BEGIN
	//проверка загруженных данных
	IF #load <> #last THEN
	    #ok := FALSE;
	END_IF;
	
	//первичная загрузка данных
	IF NOT #ok THEN
	    "KP_2_10_DB".KP[0].CMD := "KP_2_10_DB".KP[#load].CMD;
	    "KP_2_10_DB".KP[0].Mode := "KP_2_10_DB".KP[#load].Mode;
	    "KP_2_10_DB".KP[0].Status := "KP_2_10_DB".KP[#load].Status;
	    "KP_2_10_DB".KP[0].FB := "KP_2_10_DB".KP[#load].FB;
	    "KP_2_10_DB".KP[0].Use := "KP_2_10_DB".KP[#load].Use;
	    "KP_2_10_DB".KP[0].Alarm := "KP_2_10_DB".KP[#load].Alarm;
	    "KP_2_10_DB".KP[0].Clock[0].SP := "KP_2_10_DB".KP[#load].Clock[0].SP;
	    "KP_2_10_DB".KP[0].Clock[0].Now := "KP_2_10_DB".KP[#load].Clock[0].Now;
	    "KP_2_10_DB".KP[0].Clock[1].SP := "KP_2_10_DB".KP[#load].Clock[1].SP;
	    "KP_2_10_DB".KP[0].Clock[1].Now := "KP_2_10_DB".KP[#load].Clock[1].Now;
	    "KP_2_10_DB".KP[0].Clock[2].SP := "KP_2_10_DB".KP[#load].Clock[2].SP;
	    "KP_2_10_DB".KP[0].Clock[2].Now := "KP_2_10_DB".KP[#load].Clock[2].Now;
	    "KP_2_10_DB".KP[0].Clock[3].SP := "KP_2_10_DB".KP[#load].Clock[3].SP;
	    "KP_2_10_DB".KP[0].Clock[3].Now := "KP_2_10_DB".KP[#load].Clock[3].Now;
	    "KP_2_10_DB".KP[0].Clock[4].SP := "KP_2_10_DB".KP[#load].Clock[4].SP;
	    "KP_2_10_DB".KP[0].Clock[4].Now := "KP_2_10_DB".KP[#load].Clock[4].Now;
	    "KP_2_10_DB".KP[0].CodeID := "KP_2_10_DB".KP[#load].CodeID;
	    "KP_2_10_DB".KP[0].Position := "KP_2_10_DB".KP[#load].Position;
	    "KP_2_10_DB".KP[0].Speed := "KP_2_10_DB".KP[#load].Speed;
	    "KP_2_10_DB".KP[0].Name := "KP_2_10_DB".KP[#load].Name;
	    #ok := true;
	    #last := #load;
	END_IF;
	
	//управление с панели
	IF #ok THEN
	    "KP_2_10_DB".KP[#load].CMD.Hand := "KP_2_10_DB".KP[0].CMD.Hand;
	    "KP_2_10_DB".KP[#load].CMD.Force := "KP_2_10_DB".KP[0].CMD.Force;
	    "KP_2_10_DB".KP[#load].CMD.Start_M := "KP_2_10_DB".KP[0].CMD.Start_M;
	    "KP_2_10_DB".KP[#load].CMD.Reset := "KP_2_10_DB".KP[0].CMD.Reset;
	    "KP_2_10_DB".KP[#load].Use := "KP_2_10_DB".KP[0].Use;
	    "KP_2_10_DB".KP[#load].Clock[0].SP := "KP_2_10_DB".KP[0].Clock[0].SP;
	    "KP_2_10_DB".KP[#load].Clock[1].SP := "KP_2_10_DB".KP[0].Clock[1].SP;
	    "KP_2_10_DB".KP[#load].Clock[2].SP := "KP_2_10_DB".KP[0].Clock[2].SP;
	    "KP_2_10_DB".KP[#load].Clock[3].SP := "KP_2_10_DB".KP[0].Clock[3].SP;
	    "KP_2_10_DB".KP[#load].Clock[4].SP := "KP_2_10_DB".KP[0].Clock[4].SP;
	    "KP_2_10_DB".KP[#load].CodeID := "KP_2_10_DB".KP[0].CodeID;
	    "KP_2_10_DB".KP[#load].Speed := "KP_2_10_DB".KP[0].Speed;
	    "KP_2_10_DB".KP[0].CMD.Local := "KP_2_10_DB".KP[#load].CMD.Local;
	    "KP_2_10_DB".KP[0].CMD.Lock := "KP_2_10_DB".KP[#load].CMD.Lock;
	    "KP_2_10_DB".KP[0].Mode := "KP_2_10_DB".KP[#load].Mode;
	    "KP_2_10_DB".KP[0].Status := "KP_2_10_DB".KP[#load].Status;
	    "KP_2_10_DB".KP[0].FB := "KP_2_10_DB".KP[#load].FB;
	    "KP_2_10_DB".KP[0].Alarm := "KP_2_10_DB".KP[#load].Alarm;
	    "KP_2_10_DB".KP[0].Clock[0].Now := "KP_2_10_DB".KP[#load].Clock[0].Now;
	    "KP_2_10_DB".KP[0].Clock[1].Now := "KP_2_10_DB".KP[#load].Clock[1].Now;
	    "KP_2_10_DB".KP[0].Clock[2].Now := "KP_2_10_DB".KP[#load].Clock[2].Now;
	    "KP_2_10_DB".KP[0].Clock[3].Now := "KP_2_10_DB".KP[#load].Clock[3].Now;
	    "KP_2_10_DB".KP[0].Clock[4].Now := "KP_2_10_DB".KP[#load].Clock[4].Now;
	    "KP_2_10_DB".KP[0].Position := "KP_2_10_DB".KP[#load].Position;
	    IF "KP_2_10_DB".KP[0].CMD.Reset THEN
	        "KP_2_10_DB".KP[0].CMD.Reset := FALSE;
	    END_IF;
	END_IF;
	
	    
END_FUNCTION

FUNCTION_BLOCK "KP_1"
{ S7_Optimized_Access := 'FALSE' }
VERSION : 0.1
   VAR 
      limit { S7_SetPoint := 'True'} : Int := 2;   // число задвижек в камере
      load : Int;   // отображаемые на экране настройки
      load_last : Int;
      KP : Array[0..10] of "DRV_AUMA";
      load_ok { S7_SetPoint := 'True'} : Bool;
   END_VAR

   VAR_TEMP 
      ID : Int;
      cnt : Int;
   END_VAR


BEGIN
	
	"Load_KP_1"(last := #load_last,
	              load := #load,
	              ok := #load_ok);
	  IF "KP_Reset" THEN
	      #load := 10;
	  END_IF;
	
	FOR #cnt := 1 TO #limit BY 1 DO
	    #ID := #KP[#cnt].CodeID;
	    #KP[#cnt].CMD.Local := NOT "AUMA_KP_1_DB".AUMA[#ID].Message.Sel_Dist;
	    #KP[#cnt].Alarm.Link := NOT "AUMA_KP_1_DB".AUMA[#ID].Link;
	    #KP[#cnt].Use.Enable := "AUMA_KP_1_DB".AUMA[#ID].Use;
	    #KP[#cnt].Name := "AUMA_KP_1_DB".AUMA[#ID].Name;
	    #KP[#cnt].Position := INT_TO_REAL("AUMA_KP_1_DB".AUMA[#ID].Position) / 10.0;
	    #KP[#cnt].FB.QF := "AUMA_KP_1_DB".AUMA[#ID].Message.NotReady;
	    #KP[#cnt].FB.KM_Open := "AUMA_KP_1_DB".AUMA[#ID].Message.Opening;
	    #KP[#cnt].FB.KM_Close := "AUMA_KP_1_DB".AUMA[#ID].Message.Closing;
	    #KP[#cnt].FB.Open := "AUMA_KP_1_DB".AUMA[#ID].Message.Open;
	    #KP[#cnt].FB.Close := "AUMA_KP_1_DB".AUMA[#ID].Message.Close;
	    #KP[#cnt]();
	    "AUMA_KP_1_DB".AUMA[#ID].Speed := #KP[#cnt].Speed;
	    "AUMA_KP_1_DB".AUMA[#ID].CMD.Open := #KP[#cnt].CMD_Open;
	    "AUMA_KP_1_DB".AUMA[#ID].CMD.Close := #KP[#cnt].CMD_Close;
	    IF "AUMA_KP_1_DB".AUMA[#ID].CMD.Open <> "AUMA_KP_1_DB".AUMA[#ID].CMD_last.Open THEN
	        "AUMA_KP_1_DB".AUMA[#ID].CMD_last.Open := "AUMA_KP_1_DB".AUMA[#ID].CMD.Open;
	        "AUMA_KP_1_DB".AUMA[#ID].Update := true;
	    END_IF;
	    IF "AUMA_KP_1_DB".AUMA[#ID].CMD.Close <> "AUMA_KP_1_DB".AUMA[#ID].CMD_last.Close THEN
	        "AUMA_KP_1_DB".AUMA[#ID].CMD_last.Close := "AUMA_KP_1_DB".AUMA[#ID].CMD.Close;
	        "AUMA_KP_1_DB".AUMA[#ID].Update := true;
	    END_IF;
	END_FOR;
END_FUNCTION_BLOCK

FUNCTION "Load_KP_1" : Void
{ S7_Optimized_Access := 'TRUE' }
VERSION : 0.1
   VAR_IN_OUT 
      ok : Bool;
      load : Int;
      last : Int;
   END_VAR


BEGIN
	//проверка загруженных данных
	IF #load <> #last THEN
	    #ok := FALSE;
	END_IF;
	
	//первичная загрузка данных
	IF NOT #ok THEN
	    "KP_1_DB".KP[0].CMD := "KP_1_DB".KP[#load].CMD;
	    "KP_1_DB".KP[0].Mode := "KP_1_DB".KP[#load].Mode;
	    "KP_1_DB".KP[0].Status := "KP_1_DB".KP[#load].Status;
	    "KP_1_DB".KP[0].FB := "KP_1_DB".KP[#load].FB;
	    "KP_1_DB".KP[0].Use := "KP_1_DB".KP[#load].Use;
	    "KP_1_DB".KP[0].Alarm := "KP_1_DB".KP[#load].Alarm;
	    "KP_1_DB".KP[0].Clock[0].SP := "KP_1_DB".KP[#load].Clock[0].SP;
	    "KP_1_DB".KP[0].Clock[0].Now := "KP_1_DB".KP[#load].Clock[0].Now;
	    "KP_1_DB".KP[0].Clock[1].SP := "KP_1_DB".KP[#load].Clock[1].SP;
	    "KP_1_DB".KP[0].Clock[1].Now := "KP_1_DB".KP[#load].Clock[1].Now;
	    "KP_1_DB".KP[0].Clock[2].SP := "KP_1_DB".KP[#load].Clock[2].SP;
	    "KP_1_DB".KP[0].Clock[2].Now := "KP_1_DB".KP[#load].Clock[2].Now;
	    "KP_1_DB".KP[0].Clock[3].SP := "KP_1_DB".KP[#load].Clock[3].SP;
	    "KP_1_DB".KP[0].Clock[3].Now := "KP_1_DB".KP[#load].Clock[3].Now;
	    "KP_1_DB".KP[0].Clock[4].SP := "KP_1_DB".KP[#load].Clock[4].SP;
	    "KP_1_DB".KP[0].Clock[4].Now := "KP_1_DB".KP[#load].Clock[4].Now;
	    "KP_1_DB".KP[0].CodeID := "KP_1_DB".KP[#load].CodeID;
	    "KP_1_DB".KP[0].Position := "KP_1_DB".KP[#load].Position;
	    "KP_1_DB".KP[0].Speed := "KP_1_DB".KP[#load].Speed;
	    "KP_1_DB".KP[0].Name := "KP_1_DB".KP[#load].Name;
	    #ok := true;
	    #last := #load;
	END_IF;
	
	//управление с панели
	IF #ok THEN
	    "KP_1_DB".KP[#load].CMD.Hand := "KP_1_DB".KP[0].CMD.Hand;
	    "KP_1_DB".KP[#load].CMD.Force := "KP_1_DB".KP[0].CMD.Force;
	    "KP_1_DB".KP[#load].CMD.Start_M := "KP_1_DB".KP[0].CMD.Start_M;
	    "KP_1_DB".KP[#load].CMD.Reset := "KP_1_DB".KP[0].CMD.Reset;
	    "KP_1_DB".KP[#load].Use := "KP_1_DB".KP[0].Use;
	    "KP_1_DB".KP[#load].Clock[0].SP := "KP_1_DB".KP[0].Clock[0].SP;
	    "KP_1_DB".KP[#load].Clock[1].SP := "KP_1_DB".KP[0].Clock[1].SP;
	    "KP_1_DB".KP[#load].Clock[2].SP := "KP_1_DB".KP[0].Clock[2].SP;
	    "KP_1_DB".KP[#load].Clock[3].SP := "KP_1_DB".KP[0].Clock[3].SP;
	    "KP_1_DB".KP[#load].Clock[4].SP := "KP_1_DB".KP[0].Clock[4].SP;
	    "KP_1_DB".KP[#load].CodeID := "KP_1_DB".KP[0].CodeID;
	    "KP_1_DB".KP[#load].Speed := "KP_1_DB".KP[0].Speed;
	    "KP_1_DB".KP[0].CMD.Local := "KP_1_DB".KP[#load].CMD.Local;
	    "KP_1_DB".KP[0].CMD.Lock := "KP_1_DB".KP[#load].CMD.Lock;
	    "KP_1_DB".KP[0].Mode := "KP_1_DB".KP[#load].Mode;
	    "KP_1_DB".KP[0].Status := "KP_1_DB".KP[#load].Status;
	    "KP_1_DB".KP[0].FB := "KP_1_DB".KP[#load].FB;
	    "KP_1_DB".KP[0].Alarm := "KP_1_DB".KP[#load].Alarm;
	    "KP_1_DB".KP[0].Clock[0].Now := "KP_1_DB".KP[#load].Clock[0].Now;
	    "KP_1_DB".KP[0].Clock[1].Now := "KP_1_DB".KP[#load].Clock[1].Now;
	    "KP_1_DB".KP[0].Clock[2].Now := "KP_1_DB".KP[#load].Clock[2].Now;
	    "KP_1_DB".KP[0].Clock[3].Now := "KP_1_DB".KP[#load].Clock[3].Now;
	    "KP_1_DB".KP[0].Clock[4].Now := "KP_1_DB".KP[#load].Clock[4].Now;
	    "KP_1_DB".KP[0].Position := "KP_1_DB".KP[#load].Position;
	    IF "KP_1_DB".KP[0].CMD.Reset THEN
	        "KP_1_DB".KP[0].CMD.Reset := FALSE;
	    END_IF;
	END_IF;
	
	    
END_FUNCTION

FUNCTION_BLOCK "KP_2"
{ S7_Optimized_Access := 'FALSE' }
VERSION : 0.1
   VAR 
      limit { S7_SetPoint := 'True'} : Int := 2;   // число задвижек в камере
      load : Int;   // отображаемые на экране настройки
      load_last : Int;
      KP : Array[0..10] of "DRV_AUMA";
      load_ok { S7_SetPoint := 'True'} : Bool;
   END_VAR

   VAR_TEMP 
      ID : Int;
      cnt : Int;
   END_VAR


BEGIN
	
	"Load_KP_2"(last := #load_last,
	              load := #load,
	              ok := #load_ok);
	  IF "KP_Reset" THEN
	      #load := 10;
	  END_IF;
	
	FOR #cnt := 1 TO #limit BY 1 DO
	    #ID := #KP[#cnt].CodeID;
	    #KP[#cnt].CMD.Local := NOT "AUMA_KP_2_DB".AUMA[#ID].Message.Sel_Dist;
	    #KP[#cnt].Alarm.Link := NOT "AUMA_KP_2_DB".AUMA[#ID].Link;
	    #KP[#cnt].Use.Enable := "AUMA_KP_2_DB".AUMA[#ID].Use;
	    #KP[#cnt].Name := "AUMA_KP_2_DB".AUMA[#ID].Name;
	    #KP[#cnt].Position := INT_TO_REAL("AUMA_KP_2_DB".AUMA[#ID].Position) / 10.0;
	    #KP[#cnt].FB.QF := "AUMA_KP_2_DB".AUMA[#ID].Message.NotReady;
	    #KP[#cnt].FB.KM_Open := "AUMA_KP_2_DB".AUMA[#ID].Message.Opening;
	    #KP[#cnt].FB.KM_Close := "AUMA_KP_2_DB".AUMA[#ID].Message.Closing;
	    #KP[#cnt].FB.Open := "AUMA_KP_2_DB".AUMA[#ID].Message.Open;
	    #KP[#cnt].FB.Close := "AUMA_KP_2_DB".AUMA[#ID].Message.Close;
	    #KP[#cnt]();
	    "AUMA_KP_2_DB".AUMA[#ID].Speed := #KP[#cnt].Speed;
	    "AUMA_KP_2_DB".AUMA[#ID].CMD.Open := #KP[#cnt].CMD_Open;
	    "AUMA_KP_2_DB".AUMA[#ID].CMD.Close := #KP[#cnt].CMD_Close;
	    IF "AUMA_KP_2_DB".AUMA[#ID].CMD.Open <> "AUMA_KP_2_DB".AUMA[#ID].CMD_last.Open THEN
	        "AUMA_KP_2_DB".AUMA[#ID].CMD_last.Open := "AUMA_KP_2_DB".AUMA[#ID].CMD.Open;
	        "AUMA_KP_2_DB".AUMA[#ID].Update := true;
	    END_IF;
	    IF "AUMA_KP_2_DB".AUMA[#ID].CMD.Close <> "AUMA_KP_2_DB".AUMA[#ID].CMD_last.Close THEN
	        "AUMA_KP_2_DB".AUMA[#ID].CMD_last.Close := "AUMA_KP_2_DB".AUMA[#ID].CMD.Close;
	        "AUMA_KP_2_DB".AUMA[#ID].Update := true;
	    END_IF;
	END_FOR;
END_FUNCTION_BLOCK

FUNCTION "Load_KP_2" : Void
{ S7_Optimized_Access := 'TRUE' }
VERSION : 0.1
   VAR_IN_OUT 
      ok : Bool;
      load : Int;
      last : Int;
   END_VAR


BEGIN
	//проверка загруженных данных
	IF #load <> #last THEN
	    #ok := FALSE;
	END_IF;
	
	//первичная загрузка данных
	IF NOT #ok THEN
	    "KP_2_DB".KP[0].CMD := "KP_2_DB".KP[#load].CMD;
	    "KP_2_DB".KP[0].Mode := "KP_2_DB".KP[#load].Mode;
	    "KP_2_DB".KP[0].Status := "KP_2_DB".KP[#load].Status;
	    "KP_2_DB".KP[0].FB := "KP_2_DB".KP[#load].FB;
	    "KP_2_DB".KP[0].Use := "KP_2_DB".KP[#load].Use;
	    "KP_2_DB".KP[0].Alarm := "KP_2_DB".KP[#load].Alarm;
	    "KP_2_DB".KP[0].Clock[0].SP := "KP_2_DB".KP[#load].Clock[0].SP;
	    "KP_2_DB".KP[0].Clock[0].Now := "KP_2_DB".KP[#load].Clock[0].Now;
	    "KP_2_DB".KP[0].Clock[1].SP := "KP_2_DB".KP[#load].Clock[1].SP;
	    "KP_2_DB".KP[0].Clock[1].Now := "KP_2_DB".KP[#load].Clock[1].Now;
	    "KP_2_DB".KP[0].Clock[2].SP := "KP_2_DB".KP[#load].Clock[2].SP;
	    "KP_2_DB".KP[0].Clock[2].Now := "KP_2_DB".KP[#load].Clock[2].Now;
	    "KP_2_DB".KP[0].Clock[3].SP := "KP_2_DB".KP[#load].Clock[3].SP;
	    "KP_2_DB".KP[0].Clock[3].Now := "KP_2_DB".KP[#load].Clock[3].Now;
	    "KP_2_DB".KP[0].Clock[4].SP := "KP_2_DB".KP[#load].Clock[4].SP;
	    "KP_2_DB".KP[0].Clock[4].Now := "KP_2_DB".KP[#load].Clock[4].Now;
	    "KP_2_DB".KP[0].CodeID := "KP_2_DB".KP[#load].CodeID;
	    "KP_2_DB".KP[0].Position := "KP_2_DB".KP[#load].Position;
	    "KP_2_DB".KP[0].Speed := "KP_2_DB".KP[#load].Speed;
	    "KP_2_DB".KP[0].Name := "KP_2_DB".KP[#load].Name;
	    #ok := true;
	    #last := #load;
	END_IF;
	
	//управление с панели
	IF #ok THEN
	    "KP_2_DB".KP[#load].CMD.Hand := "KP_2_DB".KP[0].CMD.Hand;
	    "KP_2_DB".KP[#load].CMD.Force := "KP_2_DB".KP[0].CMD.Force;
	    "KP_2_DB".KP[#load].CMD.Start_M := "KP_2_DB".KP[0].CMD.Start_M;
	    "KP_2_DB".KP[#load].CMD.Reset := "KP_2_DB".KP[0].CMD.Reset;
	    "KP_2_DB".KP[#load].Use := "KP_2_DB".KP[0].Use;
	    "KP_2_DB".KP[#load].Clock[0].SP := "KP_2_DB".KP[0].Clock[0].SP;
	    "KP_2_DB".KP[#load].Clock[1].SP := "KP_2_DB".KP[0].Clock[1].SP;
	    "KP_2_DB".KP[#load].Clock[2].SP := "KP_2_DB".KP[0].Clock[2].SP;
	    "KP_2_DB".KP[#load].Clock[3].SP := "KP_2_DB".KP[0].Clock[3].SP;
	    "KP_2_DB".KP[#load].Clock[4].SP := "KP_2_DB".KP[0].Clock[4].SP;
	    "KP_2_DB".KP[#load].CodeID := "KP_2_DB".KP[0].CodeID;
	    "KP_2_DB".KP[#load].Speed := "KP_2_DB".KP[0].Speed;
	    "KP_2_DB".KP[0].CMD.Local := "KP_2_DB".KP[#load].CMD.Local;
	    "KP_2_DB".KP[0].CMD.Lock := "KP_2_DB".KP[#load].CMD.Lock;
	    "KP_2_DB".KP[0].Mode := "KP_2_DB".KP[#load].Mode;
	    "KP_2_DB".KP[0].Status := "KP_2_DB".KP[#load].Status;
	    "KP_2_DB".KP[0].FB := "KP_2_DB".KP[#load].FB;
	    "KP_2_DB".KP[0].Alarm := "KP_2_DB".KP[#load].Alarm;
	    "KP_2_DB".KP[0].Clock[0].Now := "KP_2_DB".KP[#load].Clock[0].Now;
	    "KP_2_DB".KP[0].Clock[1].Now := "KP_2_DB".KP[#load].Clock[1].Now;
	    "KP_2_DB".KP[0].Clock[2].Now := "KP_2_DB".KP[#load].Clock[2].Now;
	    "KP_2_DB".KP[0].Clock[3].Now := "KP_2_DB".KP[#load].Clock[3].Now;
	    "KP_2_DB".KP[0].Clock[4].Now := "KP_2_DB".KP[#load].Clock[4].Now;
	    "KP_2_DB".KP[0].Position := "KP_2_DB".KP[#load].Position;
	    IF "KP_2_DB".KP[0].CMD.Reset THEN
	        "KP_2_DB".KP[0].CMD.Reset := FALSE;
	    END_IF;
	END_IF;
	
	    
END_FUNCTION

FUNCTION_BLOCK "KP_3"
{ S7_Optimized_Access := 'FALSE' }
VERSION : 0.1
   VAR 
      limit { S7_SetPoint := 'True'} : Int := 2;   // число задвижек в камере
      load : Int;   // отображаемые на экране настройки
      load_last : Int;
      KP : Array[0..10] of "DRV_AUMA";
      load_ok { S7_SetPoint := 'True'} : Bool;
   END_VAR

   VAR_TEMP 
      ID : Int;
      cnt : Int;
   END_VAR


BEGIN
	
	"Load_KP_3"(last := #load_last,
	              load := #load,
	              ok := #load_ok);
	  IF "KP_Reset" THEN
	      #load := 10;
	  END_IF;
	
	FOR #cnt := 1 TO #limit BY 1 DO
	    #ID := #KP[#cnt].CodeID;
	    #KP[#cnt].CMD.Local := NOT "AUMA_KP_3_DB".AUMA[#ID].Message.Sel_Dist;
	    #KP[#cnt].Alarm.Link := NOT "AUMA_KP_3_DB".AUMA[#ID].Link;
	    #KP[#cnt].Use.Enable := "AUMA_KP_3_DB".AUMA[#ID].Use;
	    #KP[#cnt].Name := "AUMA_KP_3_DB".AUMA[#ID].Name;
	    #KP[#cnt].Position := INT_TO_REAL("AUMA_KP_3_DB".AUMA[#ID].Position) / 10.0;
	    #KP[#cnt].FB.QF := "AUMA_KP_3_DB".AUMA[#ID].Message.NotReady;
	    #KP[#cnt].FB.KM_Open := "AUMA_KP_3_DB".AUMA[#ID].Message.Opening;
	    #KP[#cnt].FB.KM_Close := "AUMA_KP_3_DB".AUMA[#ID].Message.Closing;
	    #KP[#cnt].FB.Open := "AUMA_KP_3_DB".AUMA[#ID].Message.Open;
	    #KP[#cnt].FB.Close := "AUMA_KP_3_DB".AUMA[#ID].Message.Close;
	    #KP[#cnt]();
	    "AUMA_KP_3_DB".AUMA[#ID].Speed := #KP[#cnt].Speed;
	    "AUMA_KP_3_DB".AUMA[#ID].CMD.Open := #KP[#cnt].CMD_Open;
	    "AUMA_KP_3_DB".AUMA[#ID].CMD.Close := #KP[#cnt].CMD_Close;
	    IF "AUMA_KP_3_DB".AUMA[#ID].CMD.Open <> "AUMA_KP_3_DB".AUMA[#ID].CMD_last.Open THEN
	        "AUMA_KP_3_DB".AUMA[#ID].CMD_last.Open := "AUMA_KP_3_DB".AUMA[#ID].CMD.Open;
	        "AUMA_KP_3_DB".AUMA[#ID].Update := true;
	    END_IF;
	    IF "AUMA_KP_3_DB".AUMA[#ID].CMD.Close <> "AUMA_KP_3_DB".AUMA[#ID].CMD_last.Close THEN
	        "AUMA_KP_3_DB".AUMA[#ID].CMD_last.Close := "AUMA_KP_3_DB".AUMA[#ID].CMD.Close;
	        "AUMA_KP_3_DB".AUMA[#ID].Update := true;
	    END_IF;
	END_FOR;
END_FUNCTION_BLOCK

FUNCTION "Load_KP_3" : Void
{ S7_Optimized_Access := 'TRUE' }
VERSION : 0.1
   VAR_IN_OUT 
      ok : Bool;
      load : Int;
      last : Int;
   END_VAR


BEGIN
	//проверка загруженных данных
	IF #load <> #last THEN
	    #ok := FALSE;
	END_IF;
	
	//первичная загрузка данных
	IF NOT #ok THEN
	    "KP_3_DB".KP[0].CMD := "KP_3_DB".KP[#load].CMD;
	    "KP_3_DB".KP[0].Mode := "KP_3_DB".KP[#load].Mode;
	    "KP_3_DB".KP[0].Status := "KP_3_DB".KP[#load].Status;
	    "KP_3_DB".KP[0].FB := "KP_3_DB".KP[#load].FB;
	    "KP_3_DB".KP[0].Use := "KP_3_DB".KP[#load].Use;
	    "KP_3_DB".KP[0].Alarm := "KP_3_DB".KP[#load].Alarm;
	    "KP_3_DB".KP[0].Clock[0].SP := "KP_3_DB".KP[#load].Clock[0].SP;
	    "KP_3_DB".KP[0].Clock[0].Now := "KP_3_DB".KP[#load].Clock[0].Now;
	    "KP_3_DB".KP[0].Clock[1].SP := "KP_3_DB".KP[#load].Clock[1].SP;
	    "KP_3_DB".KP[0].Clock[1].Now := "KP_3_DB".KP[#load].Clock[1].Now;
	    "KP_3_DB".KP[0].Clock[2].SP := "KP_3_DB".KP[#load].Clock[2].SP;
	    "KP_3_DB".KP[0].Clock[2].Now := "KP_3_DB".KP[#load].Clock[2].Now;
	    "KP_3_DB".KP[0].Clock[3].SP := "KP_3_DB".KP[#load].Clock[3].SP;
	    "KP_3_DB".KP[0].Clock[3].Now := "KP_3_DB".KP[#load].Clock[3].Now;
	    "KP_3_DB".KP[0].Clock[4].SP := "KP_3_DB".KP[#load].Clock[4].SP;
	    "KP_3_DB".KP[0].Clock[4].Now := "KP_3_DB".KP[#load].Clock[4].Now;
	    "KP_3_DB".KP[0].CodeID := "KP_3_DB".KP[#load].CodeID;
	    "KP_3_DB".KP[0].Position := "KP_3_DB".KP[#load].Position;
	    "KP_3_DB".KP[0].Speed := "KP_3_DB".KP[#load].Speed;
	    "KP_3_DB".KP[0].Name := "KP_3_DB".KP[#load].Name;
	    #ok := true;
	    #last := #load;
	END_IF;
	
	//управление с панели
	IF #ok THEN
	    "KP_3_DB".KP[#load].CMD.Hand := "KP_3_DB".KP[0].CMD.Hand;
	    "KP_3_DB".KP[#load].CMD.Force := "KP_3_DB".KP[0].CMD.Force;
	    "KP_3_DB".KP[#load].CMD.Start_M := "KP_3_DB".KP[0].CMD.Start_M;
	    "KP_3_DB".KP[#load].CMD.Reset := "KP_3_DB".KP[0].CMD.Reset;
	    "KP_3_DB".KP[#load].Use := "KP_3_DB".KP[0].Use;
	    "KP_3_DB".KP[#load].Clock[0].SP := "KP_3_DB".KP[0].Clock[0].SP;
	    "KP_3_DB".KP[#load].Clock[1].SP := "KP_3_DB".KP[0].Clock[1].SP;
	    "KP_3_DB".KP[#load].Clock[2].SP := "KP_3_DB".KP[0].Clock[2].SP;
	    "KP_3_DB".KP[#load].Clock[3].SP := "KP_3_DB".KP[0].Clock[3].SP;
	    "KP_3_DB".KP[#load].Clock[4].SP := "KP_3_DB".KP[0].Clock[4].SP;
	    "KP_3_DB".KP[#load].CodeID := "KP_3_DB".KP[0].CodeID;
	    "KP_3_DB".KP[#load].Speed := "KP_3_DB".KP[0].Speed;
	    "KP_3_DB".KP[0].CMD.Local := "KP_3_DB".KP[#load].CMD.Local;
	    "KP_3_DB".KP[0].CMD.Lock := "KP_3_DB".KP[#load].CMD.Lock;
	    "KP_3_DB".KP[0].Mode := "KP_3_DB".KP[#load].Mode;
	    "KP_3_DB".KP[0].Status := "KP_3_DB".KP[#load].Status;
	    "KP_3_DB".KP[0].FB := "KP_3_DB".KP[#load].FB;
	    "KP_3_DB".KP[0].Alarm := "KP_3_DB".KP[#load].Alarm;
	    "KP_3_DB".KP[0].Clock[0].Now := "KP_3_DB".KP[#load].Clock[0].Now;
	    "KP_3_DB".KP[0].Clock[1].Now := "KP_3_DB".KP[#load].Clock[1].Now;
	    "KP_3_DB".KP[0].Clock[2].Now := "KP_3_DB".KP[#load].Clock[2].Now;
	    "KP_3_DB".KP[0].Clock[3].Now := "KP_3_DB".KP[#load].Clock[3].Now;
	    "KP_3_DB".KP[0].Clock[4].Now := "KP_3_DB".KP[#load].Clock[4].Now;
	    "KP_3_DB".KP[0].Position := "KP_3_DB".KP[#load].Position;
	    IF "KP_3_DB".KP[0].CMD.Reset THEN
	        "KP_3_DB".KP[0].CMD.Reset := FALSE;
	    END_IF;
	END_IF;
	
	    
END_FUNCTION

FUNCTION_BLOCK "KP_4"
{ S7_Optimized_Access := 'FALSE' }
VERSION : 0.1
   VAR 
      limit { S7_SetPoint := 'True'} : Int := 2;   // число задвижек в камере
      load : Int;   // отображаемые на экране настройки
      load_last : Int;
      KP : Array[0..10] of "DRV_AUMA";
      load_ok { S7_SetPoint := 'True'} : Bool;
   END_VAR

   VAR_TEMP 
      ID : Int;
      cnt : Int;
   END_VAR


BEGIN
	
	"Load_KP_4"(last := #load_last,
	              load := #load,
	              ok := #load_ok);
	  IF "KP_Reset" THEN
	      #load := 10;
	  END_IF;
	
	FOR #cnt := 1 TO #limit BY 1 DO
	    #ID := #KP[#cnt].CodeID;
	    #KP[#cnt].CMD.Local := NOT "AUMA_KP_4_DB".AUMA[#ID].Message.Sel_Dist;
	    #KP[#cnt].Alarm.Link := NOT "AUMA_KP_4_DB".AUMA[#ID].Link;
	    #KP[#cnt].Use.Enable := "AUMA_KP_4_DB".AUMA[#ID].Use;
	    #KP[#cnt].Name := "AUMA_KP_4_DB".AUMA[#ID].Name;
	    #KP[#cnt].Position := INT_TO_REAL("AUMA_KP_4_DB".AUMA[#ID].Position) / 10.0;
	    #KP[#cnt].FB.QF := "AUMA_KP_4_DB".AUMA[#ID].Message.NotReady;
	    #KP[#cnt].FB.KM_Open := "AUMA_KP_4_DB".AUMA[#ID].Message.Opening;
	    #KP[#cnt].FB.KM_Close := "AUMA_KP_4_DB".AUMA[#ID].Message.Closing;
	    #KP[#cnt].FB.Open := "AUMA_KP_4_DB".AUMA[#ID].Message.Open;
	    #KP[#cnt].FB.Close := "AUMA_KP_4_DB".AUMA[#ID].Message.Close;
	    #KP[#cnt]();
	    "AUMA_KP_4_DB".AUMA[#ID].Speed := #KP[#cnt].Speed;
	    "AUMA_KP_4_DB".AUMA[#ID].CMD.Open := #KP[#cnt].CMD_Open;
	    "AUMA_KP_4_DB".AUMA[#ID].CMD.Close := #KP[#cnt].CMD_Close;
	    IF "AUMA_KP_4_DB".AUMA[#ID].CMD.Open <> "AUMA_KP_4_DB".AUMA[#ID].CMD_last.Open THEN
	        "AUMA_KP_4_DB".AUMA[#ID].CMD_last.Open := "AUMA_KP_4_DB".AUMA[#ID].CMD.Open;
	        "AUMA_KP_4_DB".AUMA[#ID].Update := true;
	    END_IF;
	    IF "AUMA_KP_4_DB".AUMA[#ID].CMD.Close <> "AUMA_KP_4_DB".AUMA[#ID].CMD_last.Close THEN
	        "AUMA_KP_4_DB".AUMA[#ID].CMD_last.Close := "AUMA_KP_4_DB".AUMA[#ID].CMD.Close;
	        "AUMA_KP_4_DB".AUMA[#ID].Update := true;
	    END_IF;
	END_FOR;
END_FUNCTION_BLOCK

FUNCTION "Load_KP_4" : Void
{ S7_Optimized_Access := 'TRUE' }
VERSION : 0.1
   VAR_IN_OUT 
      ok : Bool;
      load : Int;
      last : Int;
   END_VAR


BEGIN
	//проверка загруженных данных
	IF #load <> #last THEN
	    #ok := FALSE;
	END_IF;
	
	//первичная загрузка данных
	IF NOT #ok THEN
	    "KP_4_DB".KP[0].CMD := "KP_4_DB".KP[#load].CMD;
	    "KP_4_DB".KP[0].Mode := "KP_4_DB".KP[#load].Mode;
	    "KP_4_DB".KP[0].Status := "KP_4_DB".KP[#load].Status;
	    "KP_4_DB".KP[0].FB := "KP_4_DB".KP[#load].FB;
	    "KP_4_DB".KP[0].Use := "KP_4_DB".KP[#load].Use;
	    "KP_4_DB".KP[0].Alarm := "KP_4_DB".KP[#load].Alarm;
	    "KP_4_DB".KP[0].Clock[0].SP := "KP_4_DB".KP[#load].Clock[0].SP;
	    "KP_4_DB".KP[0].Clock[0].Now := "KP_4_DB".KP[#load].Clock[0].Now;
	    "KP_4_DB".KP[0].Clock[1].SP := "KP_4_DB".KP[#load].Clock[1].SP;
	    "KP_4_DB".KP[0].Clock[1].Now := "KP_4_DB".KP[#load].Clock[1].Now;
	    "KP_4_DB".KP[0].Clock[2].SP := "KP_4_DB".KP[#load].Clock[2].SP;
	    "KP_4_DB".KP[0].Clock[2].Now := "KP_4_DB".KP[#load].Clock[2].Now;
	    "KP_4_DB".KP[0].Clock[3].SP := "KP_4_DB".KP[#load].Clock[3].SP;
	    "KP_4_DB".KP[0].Clock[3].Now := "KP_4_DB".KP[#load].Clock[3].Now;
	    "KP_4_DB".KP[0].Clock[4].SP := "KP_4_DB".KP[#load].Clock[4].SP;
	    "KP_4_DB".KP[0].Clock[4].Now := "KP_4_DB".KP[#load].Clock[4].Now;
	    "KP_4_DB".KP[0].CodeID := "KP_4_DB".KP[#load].CodeID;
	    "KP_4_DB".KP[0].Position := "KP_4_DB".KP[#load].Position;
	    "KP_4_DB".KP[0].Speed := "KP_4_DB".KP[#load].Speed;
	    "KP_4_DB".KP[0].Name := "KP_4_DB".KP[#load].Name;
	    #ok := true;
	    #last := #load;
	END_IF;
	
	//управление с панели
	IF #ok THEN
	    "KP_4_DB".KP[#load].CMD.Hand := "KP_4_DB".KP[0].CMD.Hand;
	    "KP_4_DB".KP[#load].CMD.Force := "KP_4_DB".KP[0].CMD.Force;
	    "KP_4_DB".KP[#load].CMD.Start_M := "KP_4_DB".KP[0].CMD.Start_M;
	    "KP_4_DB".KP[#load].CMD.Reset := "KP_4_DB".KP[0].CMD.Reset;
	    "KP_4_DB".KP[#load].Use := "KP_4_DB".KP[0].Use;
	    "KP_4_DB".KP[#load].Clock[0].SP := "KP_4_DB".KP[0].Clock[0].SP;
	    "KP_4_DB".KP[#load].Clock[1].SP := "KP_4_DB".KP[0].Clock[1].SP;
	    "KP_4_DB".KP[#load].Clock[2].SP := "KP_4_DB".KP[0].Clock[2].SP;
	    "KP_4_DB".KP[#load].Clock[3].SP := "KP_4_DB".KP[0].Clock[3].SP;
	    "KP_4_DB".KP[#load].Clock[4].SP := "KP_4_DB".KP[0].Clock[4].SP;
	    "KP_4_DB".KP[#load].CodeID := "KP_4_DB".KP[0].CodeID;
	    "KP_4_DB".KP[#load].Speed := "KP_4_DB".KP[0].Speed;
	    "KP_4_DB".KP[0].CMD.Local := "KP_4_DB".KP[#load].CMD.Local;
	    "KP_4_DB".KP[0].CMD.Lock := "KP_4_DB".KP[#load].CMD.Lock;
	    "KP_4_DB".KP[0].Mode := "KP_4_DB".KP[#load].Mode;
	    "KP_4_DB".KP[0].Status := "KP_4_DB".KP[#load].Status;
	    "KP_4_DB".KP[0].FB := "KP_4_DB".KP[#load].FB;
	    "KP_4_DB".KP[0].Alarm := "KP_4_DB".KP[#load].Alarm;
	    "KP_4_DB".KP[0].Clock[0].Now := "KP_4_DB".KP[#load].Clock[0].Now;
	    "KP_4_DB".KP[0].Clock[1].Now := "KP_4_DB".KP[#load].Clock[1].Now;
	    "KP_4_DB".KP[0].Clock[2].Now := "KP_4_DB".KP[#load].Clock[2].Now;
	    "KP_4_DB".KP[0].Clock[3].Now := "KP_4_DB".KP[#load].Clock[3].Now;
	    "KP_4_DB".KP[0].Clock[4].Now := "KP_4_DB".KP[#load].Clock[4].Now;
	    "KP_4_DB".KP[0].Position := "KP_4_DB".KP[#load].Position;
	    IF "KP_4_DB".KP[0].CMD.Reset THEN
	        "KP_4_DB".KP[0].CMD.Reset := FALSE;
	    END_IF;
	END_IF;
	
	    
END_FUNCTION

FUNCTION_BLOCK "KP_5"
{ S7_Optimized_Access := 'FALSE' }
VERSION : 0.1
   VAR 
      limit { S7_SetPoint := 'True'} : Int := 2;   // число задвижек в камере
      load : Int;   // отображаемые на экране настройки
      load_last : Int;
      KP : Array[0..10] of "DRV_AUMA";
      load_ok { S7_SetPoint := 'True'} : Bool;
   END_VAR

   VAR_TEMP 
      ID : Int;
      cnt : Int;
   END_VAR


BEGIN
	
	"Load_KP_5"(last := #load_last,
	              load := #load,
	              ok := #load_ok);
	  IF "KP_Reset" THEN
	      #load := 10;
	  END_IF;
	
	FOR #cnt := 1 TO #limit BY 1 DO
	    #ID := #KP[#cnt].CodeID;
	    #KP[#cnt].CMD.Local := NOT "AUMA_KP_5_DB".AUMA[#ID].Message.Sel_Dist;
	    #KP[#cnt].Alarm.Link := NOT "AUMA_KP_5_DB".AUMA[#ID].Link;
	    #KP[#cnt].Use.Enable := "AUMA_KP_5_DB".AUMA[#ID].Use;
	    #KP[#cnt].Name := "AUMA_KP_5_DB".AUMA[#ID].Name;
	    #KP[#cnt].Position := INT_TO_REAL("AUMA_KP_5_DB".AUMA[#ID].Position) / 10.0;
	    #KP[#cnt].FB.QF := "AUMA_KP_5_DB".AUMA[#ID].Message.NotReady;
	    #KP[#cnt].FB.KM_Open := "AUMA_KP_5_DB".AUMA[#ID].Message.Opening;
	    #KP[#cnt].FB.KM_Close := "AUMA_KP_5_DB".AUMA[#ID].Message.Closing;
	    #KP[#cnt].FB.Open := "AUMA_KP_5_DB".AUMA[#ID].Message.Open;
	    #KP[#cnt].FB.Close := "AUMA_KP_5_DB".AUMA[#ID].Message.Close;
	    #KP[#cnt]();
	    "AUMA_KP_5_DB".AUMA[#ID].Speed := #KP[#cnt].Speed;
	    "AUMA_KP_5_DB".AUMA[#ID].CMD.Open := #KP[#cnt].CMD_Open;
	    "AUMA_KP_5_DB".AUMA[#ID].CMD.Close := #KP[#cnt].CMD_Close;
	    IF "AUMA_KP_5_DB".AUMA[#ID].CMD.Open <> "AUMA_KP_5_DB".AUMA[#ID].CMD_last.Open THEN
	        "AUMA_KP_5_DB".AUMA[#ID].CMD_last.Open := "AUMA_KP_5_DB".AUMA[#ID].CMD.Open;
	        "AUMA_KP_5_DB".AUMA[#ID].Update := true;
	    END_IF;
	    IF "AUMA_KP_5_DB".AUMA[#ID].CMD.Close <> "AUMA_KP_5_DB".AUMA[#ID].CMD_last.Close THEN
	        "AUMA_KP_5_DB".AUMA[#ID].CMD_last.Close := "AUMA_KP_5_DB".AUMA[#ID].CMD.Close;
	        "AUMA_KP_5_DB".AUMA[#ID].Update := true;
	    END_IF;
	END_FOR;
END_FUNCTION_BLOCK

FUNCTION "Load_KP_5" : Void
{ S7_Optimized_Access := 'TRUE' }
VERSION : 0.1
   VAR_IN_OUT 
      ok : Bool;
      load : Int;
      last : Int;
   END_VAR


BEGIN
	//проверка загруженных данных
	IF #load <> #last THEN
	    #ok := FALSE;
	END_IF;
	
	//первичная загрузка данных
	IF NOT #ok THEN
	    "KP_5_DB".KP[0].CMD := "KP_5_DB".KP[#load].CMD;
	    "KP_5_DB".KP[0].Mode := "KP_5_DB".KP[#load].Mode;
	    "KP_5_DB".KP[0].Status := "KP_5_DB".KP[#load].Status;
	    "KP_5_DB".KP[0].FB := "KP_5_DB".KP[#load].FB;
	    "KP_5_DB".KP[0].Use := "KP_5_DB".KP[#load].Use;
	    "KP_5_DB".KP[0].Alarm := "KP_5_DB".KP[#load].Alarm;
	    "KP_5_DB".KP[0].Clock[0].SP := "KP_5_DB".KP[#load].Clock[0].SP;
	    "KP_5_DB".KP[0].Clock[0].Now := "KP_5_DB".KP[#load].Clock[0].Now;
	    "KP_5_DB".KP[0].Clock[1].SP := "KP_5_DB".KP[#load].Clock[1].SP;
	    "KP_5_DB".KP[0].Clock[1].Now := "KP_5_DB".KP[#load].Clock[1].Now;
	    "KP_5_DB".KP[0].Clock[2].SP := "KP_5_DB".KP[#load].Clock[2].SP;
	    "KP_5_DB".KP[0].Clock[2].Now := "KP_5_DB".KP[#load].Clock[2].Now;
	    "KP_5_DB".KP[0].Clock[3].SP := "KP_5_DB".KP[#load].Clock[3].SP;
	    "KP_5_DB".KP[0].Clock[3].Now := "KP_5_DB".KP[#load].Clock[3].Now;
	    "KP_5_DB".KP[0].Clock[4].SP := "KP_5_DB".KP[#load].Clock[4].SP;
	    "KP_5_DB".KP[0].Clock[4].Now := "KP_5_DB".KP[#load].Clock[4].Now;
	    "KP_5_DB".KP[0].CodeID := "KP_5_DB".KP[#load].CodeID;
	    "KP_5_DB".KP[0].Position := "KP_5_DB".KP[#load].Position;
	    "KP_5_DB".KP[0].Speed := "KP_5_DB".KP[#load].Speed;
	    "KP_5_DB".KP[0].Name := "KP_5_DB".KP[#load].Name;
	    #ok := true;
	    #last := #load;
	END_IF;
	
	//управление с панели
	IF #ok THEN
	    "KP_5_DB".KP[#load].CMD.Hand := "KP_5_DB".KP[0].CMD.Hand;
	    "KP_5_DB".KP[#load].CMD.Force := "KP_5_DB".KP[0].CMD.Force;
	    "KP_5_DB".KP[#load].CMD.Start_M := "KP_5_DB".KP[0].CMD.Start_M;
	    "KP_5_DB".KP[#load].CMD.Reset := "KP_5_DB".KP[0].CMD.Reset;
	    "KP_5_DB".KP[#load].Use := "KP_5_DB".KP[0].Use;
	    "KP_5_DB".KP[#load].Clock[0].SP := "KP_5_DB".KP[0].Clock[0].SP;
	    "KP_5_DB".KP[#load].Clock[1].SP := "KP_5_DB".KP[0].Clock[1].SP;
	    "KP_5_DB".KP[#load].Clock[2].SP := "KP_5_DB".KP[0].Clock[2].SP;
	    "KP_5_DB".KP[#load].Clock[3].SP := "KP_5_DB".KP[0].Clock[3].SP;
	    "KP_5_DB".KP[#load].Clock[4].SP := "KP_5_DB".KP[0].Clock[4].SP;
	    "KP_5_DB".KP[#load].CodeID := "KP_5_DB".KP[0].CodeID;
	    "KP_5_DB".KP[#load].Speed := "KP_5_DB".KP[0].Speed;
	    "KP_5_DB".KP[0].CMD.Local := "KP_5_DB".KP[#load].CMD.Local;
	    "KP_5_DB".KP[0].CMD.Lock := "KP_5_DB".KP[#load].CMD.Lock;
	    "KP_5_DB".KP[0].Mode := "KP_5_DB".KP[#load].Mode;
	    "KP_5_DB".KP[0].Status := "KP_5_DB".KP[#load].Status;
	    "KP_5_DB".KP[0].FB := "KP_5_DB".KP[#load].FB;
	    "KP_5_DB".KP[0].Alarm := "KP_5_DB".KP[#load].Alarm;
	    "KP_5_DB".KP[0].Clock[0].Now := "KP_5_DB".KP[#load].Clock[0].Now;
	    "KP_5_DB".KP[0].Clock[1].Now := "KP_5_DB".KP[#load].Clock[1].Now;
	    "KP_5_DB".KP[0].Clock[2].Now := "KP_5_DB".KP[#load].Clock[2].Now;
	    "KP_5_DB".KP[0].Clock[3].Now := "KP_5_DB".KP[#load].Clock[3].Now;
	    "KP_5_DB".KP[0].Clock[4].Now := "KP_5_DB".KP[#load].Clock[4].Now;
	    "KP_5_DB".KP[0].Position := "KP_5_DB".KP[#load].Position;
	    IF "KP_5_DB".KP[0].CMD.Reset THEN
	        "KP_5_DB".KP[0].CMD.Reset := FALSE;
	    END_IF;
	END_IF;
	
	    
END_FUNCTION

FUNCTION_BLOCK "PIDx"   // FB260, LAD
{ S7_Optimized_Access := 'TRUE' }
VERSION : 0.1
// stored: AutoNumber false, IsIECCheckEnabled false, IsRetainMemResEnabled false, MemoryReserve 100, SetENOAutomatically false, UDAEnableTagReadback false
   VAR DB_SPECIFIC
      Time_DTL { S7_SetPoint := 'True'} : DTL;
   END_VAR
BEGIN

REGION Network 2: Метка времени
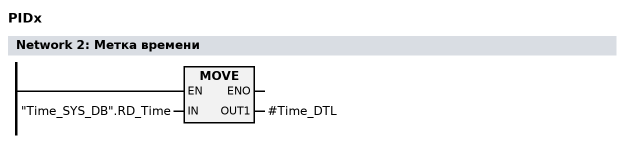
   RUNG wire#powerrail
      Move(in := "Time_SYS_DB".RD_Time, out1 => #Time_DTL)
   END_RUNG
   // the same network as SCL:
   #Time_DTL := "Time_SYS_DB".RD_Time;
END_REGION
END_FUNCTION_BLOCK

FUNCTION_BLOCK "DOx_1"   // FB210, LAD
{ S7_Optimized_Access := 'FALSE' }
VERSION : 0.1
// Start - управляющий сигнал из программы
// Q - выходной сигнал контроллера
// pulse - кратность времени в импульсном режиме
// stored: AutoNumber false, IsIECCheckEnabled false, SetENOAutomatically false, UDAEnableTagReadback false
   VAR
      All_Alarm { S7_SetPoint := 'True'} : "DO_ex";   // Общая авария
      command_2 { S7_SetPoint := 'True'} : "DO_ex";
      command_3 { S7_SetPoint := 'True'} : "DO_ex";
      command_4 { S7_SetPoint := 'True'} : "DO_ex";
      command_5 { S7_SetPoint := 'True'} : "DO_ex";
      command_6 { S7_SetPoint := 'True'} : "DO_ex";
      command_7 { S7_SetPoint := 'True'} : "DO_ex";
      command_8 { S7_SetPoint := 'True'} : "DO_ex";
      command_9 { S7_SetPoint := 'True'} : "DO_ex";
      command_10 { S7_SetPoint := 'True'} : "DO_ex";
      command_11 { S7_SetPoint := 'True'} : "DO_ex";
      command_12 { S7_SetPoint := 'True'} : "DO_ex";
   END_VAR
   VAR DB_SPECIFIC
      Time_DTL { S7_SetPoint := 'True'} : DTL;
   END_VAR
   VAR_TEMP   // added for the SCL form of the ladder/FBD networks
      _w1 : Bool;
   END_VAR
BEGIN

REGION Network 1
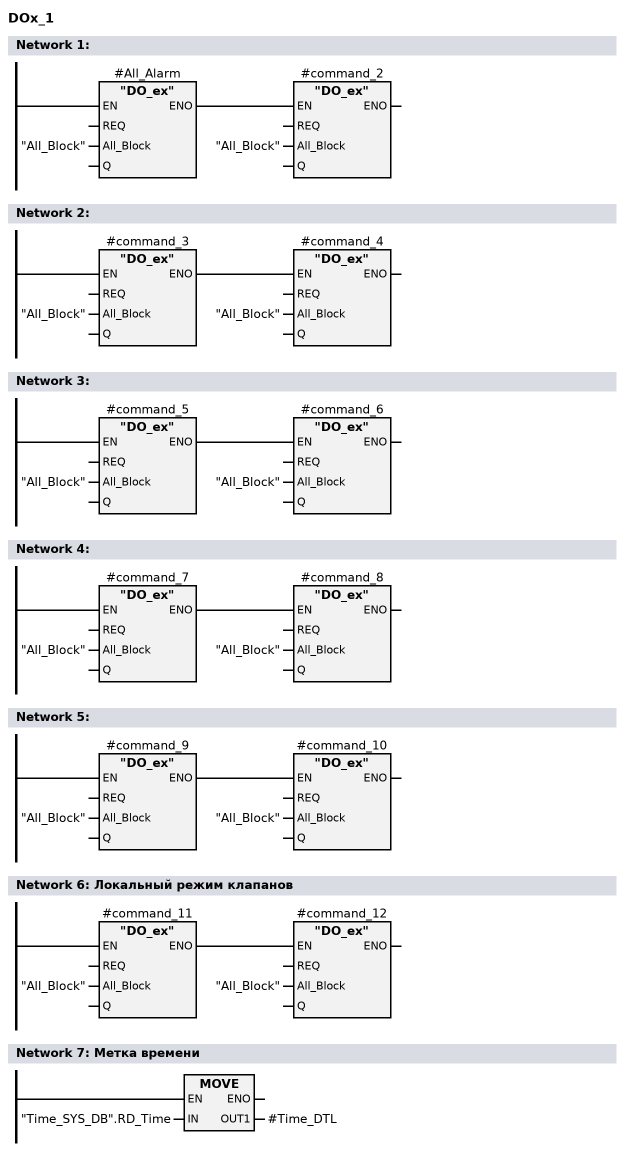
   RUNG wire#powerrail
      #All_Alarm(REQ :=, All_Block := "All_Block", Q :=)
      #command_2(REQ :=, All_Block := "All_Block", Q :=)
   END_RUNG
   // the same network as SCL:
   #All_Alarm(All_Block := "All_Block", ENO => #_w1);   // "DO_ex"
   IF #_w1 THEN
       #command_2(All_Block := "All_Block");   // "DO_ex"
   END_IF;
END_REGION

REGION Network 2
   RUNG wire#powerrail
      #command_3(REQ :=, All_Block := "All_Block", Q :=)
      #command_4(REQ :=, All_Block := "All_Block", Q :=)
   END_RUNG
   // the same network as SCL:
   #command_3(All_Block := "All_Block", ENO => #_w1);   // "DO_ex"
   IF #_w1 THEN
       #command_4(All_Block := "All_Block");   // "DO_ex"
   END_IF;
END_REGION

REGION Network 3
   RUNG wire#powerrail
      #command_5(REQ :=, All_Block := "All_Block", Q :=)
      #command_6(REQ :=, All_Block := "All_Block", Q :=)
   END_RUNG
   // the same network as SCL:
   #command_5(All_Block := "All_Block", ENO => #_w1);   // "DO_ex"
   IF #_w1 THEN
       #command_6(All_Block := "All_Block");   // "DO_ex"
   END_IF;
END_REGION

REGION Network 4
   RUNG wire#powerrail
      #command_7(REQ :=, All_Block := "All_Block", Q :=)
      #command_8(REQ :=, All_Block := "All_Block", Q :=)
   END_RUNG
   // the same network as SCL:
   #command_7(All_Block := "All_Block", ENO => #_w1);   // "DO_ex"
   IF #_w1 THEN
       #command_8(All_Block := "All_Block");   // "DO_ex"
   END_IF;
END_REGION

REGION Network 5
   RUNG wire#powerrail
      #command_9(REQ :=, All_Block := "All_Block", Q :=)
      #command_10(REQ :=, All_Block := "All_Block", Q :=)
   END_RUNG
   // the same network as SCL:
   #command_9(All_Block := "All_Block", ENO => #_w1);   // "DO_ex"
   IF #_w1 THEN
       #command_10(All_Block := "All_Block");   // "DO_ex"
   END_IF;
END_REGION

REGION Network 6: Локальный режим клапанов
   RUNG wire#powerrail
      #command_11(REQ :=, All_Block := "All_Block", Q :=)
      #command_12(REQ :=, All_Block := "All_Block", Q :=)
   END_RUNG
   // the same network as SCL:
   #command_11(All_Block := "All_Block", ENO => #_w1);   // "DO_ex"
   IF #_w1 THEN
       #command_12(All_Block := "All_Block");   // "DO_ex"
   END_IF;
END_REGION

REGION Network 7: Метка времени
   RUNG wire#powerrail
      Move(in := "Time_SYS_DB".RD_Time, out1 => #Time_DTL)
   END_RUNG
   // the same network as SCL:
   #Time_DTL := "Time_SYS_DB".RD_Time;
END_REGION
END_FUNCTION_BLOCK

FUNCTION_BLOCK "DO_ex"   // FB102, LAD
{ S7_Optimized_Access := 'FALSE' }
VERSION : 0.1
// stored: AutoNumber false, IsIECCheckEnabled false, SetENOAutomatically false, UDAEnableTagReadback false
   VAR_INPUT
      REQ : Bool;   // Запрос включения
      All_Block : Bool;
   END_VAR
   VAR_IN_OUT
      Q : Bool;   // Выходной сигнал ПЛК
   END_VAR
   VAR DB_SPECIFIC
      CMD : "CMD";   // Основные команды / Блок команд
      Use : Struct   // Функционал
         Inverse { S7_SetPoint := 'True'} : Bool;   // Инверсия входного сигнала
         Indirect { S7_SetPoint := 'True'} : Bool := true;   // Использование косвенной адресации
         Impulse { S7_SetPoint := 'True'} : Bool;   // Использовать импульсный режим
      END_STRUCT;
      ADDR_Byte { S7_SetPoint := 'True'} : Int;   // Адрес входа на контроллере (Байт)
      ADDR_Bit { S7_SetPoint := 'True'} : Int := 9;   // Адрес входа на контроллере (Бит)
      Mode : Int;
      Status : Int;
   END_VAR
   VAR
      T_Impulse { S7_SetPoint := 'True'} : "Time_S_b";   // Длительность импульса
   END_VAR
   VAR_TEMP
      Start : Bool;
   END_VAR
   VAR_TEMP   // added for the SCL form of the ladder/FBD networks
      _w1 : Bool;
   END_VAR
BEGIN

REGION Network 1: Устройство в ручном режиме
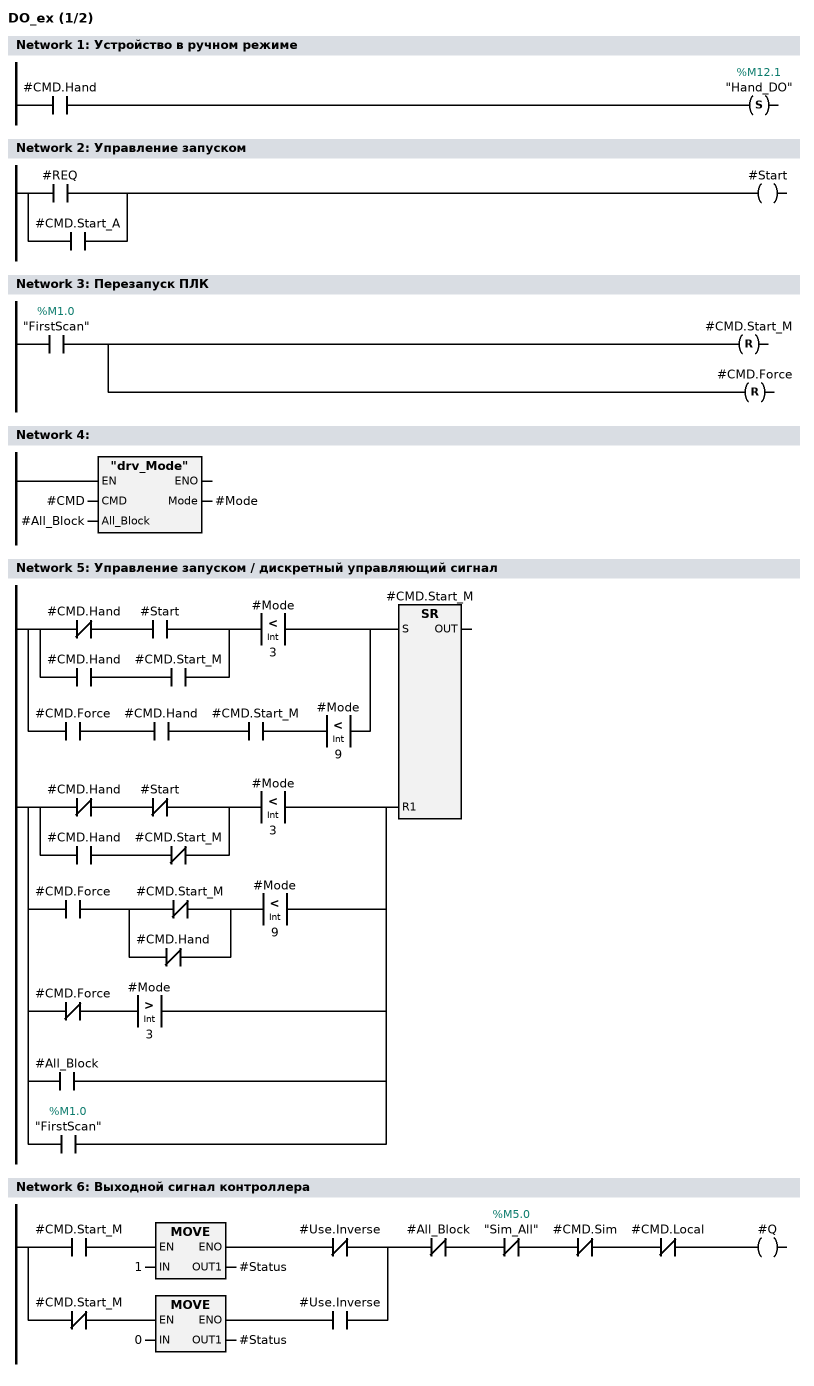
   RUNG wire#powerrail
      Contact( #CMD.Hand )
      S_Coil( "Hand_DO" )
   END_RUNG
   // the same network as SCL:
   IF #CMD.Hand THEN "Hand_DO" := TRUE; END_IF;
END_REGION

REGION Network 2: Управление запуском
   RUNG wire#powerrail
      Contact( #REQ )
      wire#w1
      Coil( #Start )
   END_RUNG
   RUNG wire#powerrail
      Contact( #CMD.Start_A )
   END_RUNG wire#w1
   // the same network as SCL:
   #Start := #REQ OR #CMD.Start_A;
END_REGION

REGION Network 3: Перезапуск ПЛК
   RUNG wire#powerrail
      Contact( "FirstScan" )
      wire#w1
      R_Coil( #CMD.Start_M )
   END_RUNG
   RUNG wire#w1
      R_Coil( #CMD.Force )
   END_RUNG
   // the same network as SCL:
   IF "FirstScan" THEN
       #CMD.Start_M := FALSE;
       #CMD.Force := FALSE;
   END_IF;
END_REGION

REGION Network 4
   RUNG wire#powerrail
      "drv_Mode"(CMD := #CMD, All_Block := #All_Block, Mode => #Mode)
   END_RUNG
   // the same network as SCL:
   "drv_Mode"(CMD := #CMD, All_Block := #All_Block, Mode => #Mode);
END_REGION

REGION Network 5: Управление запуском / дискретный управляющий сигнал
   RUNG wire#powerrail
      I_Contact( #CMD.Hand )
      Contact( #Start )
      wire#w1
      { S7_Templates := "SrcType := Int" } LT_Contact(in1 := #Mode, in2 := 3)
      wire#w2
      S_SR(operand := #CMD.Start_M, r1 := wire#w6)
   END_RUNG
   RUNG wire#powerrail
      Contact( #CMD.Hand )
      Contact( #CMD.Start_M )
   END_RUNG wire#w1
   RUNG wire#powerrail
      Contact( #CMD.Force )
      Contact( #CMD.Hand )
      Contact( #CMD.Start_M )
      { S7_Templates := "SrcType := Int" } LT_Contact(in1 := #Mode, in2 := 9)
   END_RUNG wire#w2
   RUNG wire#powerrail
      I_Contact( #CMD.Hand )
      I_Contact( #Start )
      wire#w3
      { S7_Templates := "SrcType := Int" } LT_Contact(in1 := #Mode, in2 := 3)
   END_RUNG wire#w6
   RUNG wire#powerrail
      Contact( #CMD.Hand )
      I_Contact( #CMD.Start_M )
   END_RUNG wire#w3
   RUNG wire#powerrail
      Contact( #CMD.Force )
      wire#w4
      I_Contact( #CMD.Start_M )
      wire#w5
      { S7_Templates := "SrcType := Int" } LT_Contact(in1 := #Mode, in2 := 9)
   END_RUNG wire#w6
   RUNG wire#w4
      I_Contact( #CMD.Hand )
   END_RUNG wire#w5
   RUNG wire#powerrail
      I_Contact( #CMD.Force )
      { S7_Templates := "SrcType := Int" } GT_Contact(in1 := #Mode, in2 := 3)
   END_RUNG wire#w6
   RUNG wire#powerrail
      Contact( #All_Block )
   END_RUNG wire#w6
   RUNG wire#powerrail
      Contact( "FirstScan" )
   END_RUNG wire#w6
   // the same network as SCL:
   #_w1 := (((NOT #CMD.Hand AND NOT #Start) OR (#CMD.Hand AND NOT #CMD.Start_M)) AND (#Mode < 3)) OR (#CMD.Force AND (NOT #CMD.Start_M OR NOT #CMD.Hand) AND (#Mode < 9)) OR (NOT #CMD.Force AND (#Mode > 3)) OR #All_Block OR "FirstScan";
   IF (((NOT #CMD.Hand AND #Start) OR (#CMD.Hand AND #CMD.Start_M)) AND (#Mode < 3)) OR (#CMD.Force AND #CMD.Hand AND #CMD.Start_M AND (#Mode < 9)) THEN
       #CMD.Start_M := TRUE;   // SR flip-flop
   END_IF;
   IF #_w1 THEN #CMD.Start_M := FALSE; END_IF;
END_REGION

REGION Network 6: Выходной сигнал контроллера
   RUNG wire#powerrail
      Contact( #CMD.Start_M )
      Move(in := 1, out1 => #Status)
      I_Contact( #Use.Inverse )
      wire#w1
      I_Contact( #All_Block )
      I_Contact( "Sim_All" )
      I_Contact( #CMD.Sim )
      I_Contact( #CMD.Local )
      Coil( #Q )
   END_RUNG
   RUNG wire#powerrail
      I_Contact( #CMD.Start_M )
      Move(in := 0, out1 => #Status)
      Contact( #Use.Inverse )
   END_RUNG wire#w1
   // the same network as SCL:
   IF #CMD.Start_M THEN #Status := 1; END_IF;
   IF NOT #CMD.Start_M THEN #Status := 0; END_IF;
   #Q := ((#CMD.Start_M AND NOT #Use.Inverse) OR (NOT #CMD.Start_M AND #Use.Inverse)) AND NOT #All_Block AND NOT "Sim_All" AND NOT #CMD.Sim AND NOT #CMD.Local;
END_REGION

REGION Network 7: Косвенная адресация
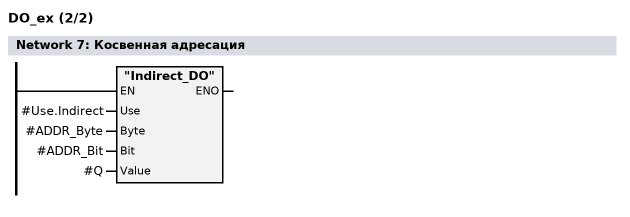
   RUNG wire#powerrail
      "Indirect_DO"(Use := #Use.Indirect, "Byte" := #ADDR_Byte, Bit := #ADDR_Bit, Value := #Q)
   END_RUNG
   // the same network as SCL:
   "Indirect_DO"(Use := #Use.Indirect, "Byte" := #ADDR_Byte, Bit := #ADDR_Bit, Value := #Q);
END_REGION
END_FUNCTION_BLOCK

FUNCTION_BLOCK "AOx"   // FB230, LAD
TITLE = Регулируемые устройства
{ S7_Optimized_Access := 'FALSE' }
VERSION : 0.1
// SP - управляющий сигнал из программы, формат Real
// Signal - PQW код выходного сигнала контроллера
// stored: AutoNumber false, IsIECCheckEnabled false, SetENOAutomatically false, UDAEnableTagReadback false
   VAR DB_SPECIFIC
      Time_DTL { S7_SetPoint := 'True'} : DTL;
   END_VAR
BEGIN

REGION Network 1: Example
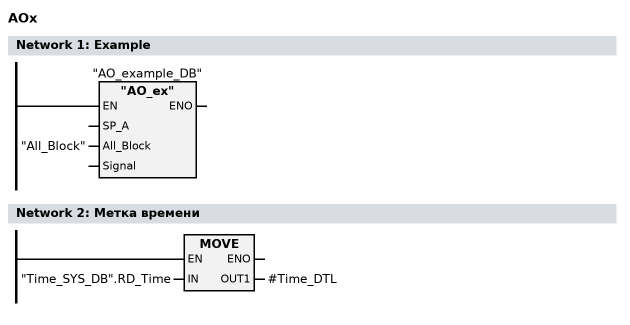
   RUNG wire#powerrail
      "AO_example_DB"(SP_A :=, All_Block := "All_Block", Signal :=)
   END_RUNG
   // the same network as SCL:
   "AO_example_DB"(All_Block := "All_Block");   // "AO_ex"
END_REGION

REGION Network 2: Метка времени
   RUNG wire#powerrail
      Move(in := "Time_SYS_DB".RD_Time, out1 => #Time_DTL)
   END_RUNG
   // the same network as SCL:
   #Time_DTL := "Time_SYS_DB".RD_Time;
END_REGION
END_FUNCTION_BLOCK

FUNCTION_BLOCK "AO_ex"   // FB104, LAD
{ S7_Optimized_Access := 'FALSE' }
VERSION : 0.1
// stored: AutoNumber false, IsIECCheckEnabled false, SetENOAutomatically false, UDAEnableTagReadback false
   VAR_INPUT
      SP_A : Real;   // Уставка авторежима
      All_Block : Bool;   // Аварийная остановка
   END_VAR
   VAR_IN_OUT
      Signal : Int;   // Входной сигнал контроллера
   END_VAR
   VAR DB_SPECIFIC
      CMD : "CMD";   // Основные команды / Блок команд
      Mode : Int;   // Режим работы
      Status : Int;   // Статус устройства
      Use : Struct   // Функционал
         Indirect { S7_SetPoint := 'True'} : Bool := true;   // Косвенная адресация
      END_STRUCT;
      VmA : Real;   // Реальный сигнал на входе ПЛК
      SP_M : Real;   // Уставка в ручном режиме
   END_VAR
   VAR
      Converter { S7_SetPoint := 'True'} : "Converter_LAD";   // Масштабирование сигнала
   END_VAR
   VAR DB_SPECIFIC
      Events : Word;   // События датчика
      pos : Array[0..15] of Bool;   // Контроль фронтов событий
      Output_Type { S7_SetPoint := 'True'} : Int;   // Тип выхода, 0 - 4..20, 1 - 0..20, 2 - 0..10, 3 - 0..5
      CodeID { S7_SetPoint := 'True'} : Int;   // Код датчика для привязки в скаде
      "Type" { S7_SetPoint := 'True'} : Int;   // Тип датчика (единицы измерения)
      ADDR { S7_SetPoint := 'True'} : Int;   // Адрес выхода на контроллере
   END_VAR
   VAR
      Slow { S7_SetPoint := 'True'} : "Slow";   // Плавное управление
   END_VAR
   VAR DB_SPECIFIC
      Time_DTL { S7_SetPoint := 'True'} : DTL;
   END_VAR
   VAR_TEMP
      ev : Bool;   // флаг управления событиями
      Signal_R : Real;   // Актуальный сигнал
      Signal_Ex : Real;   // Конвертация сигнала
      Signal_Dint : DInt;   // Сигнал в DInt
      Type_Min : Real;
      Type_Max : Real;
   END_VAR
   // CMD.Start_A := true;
   VAR_TEMP   // added for the SCL form of the ladder/FBD networks
      _w1 : Bool;
      _w2 : Bool;
      _w3 : Bool;
      _w4 : Bool;
      _w5 : Bool;
      _w6 : Bool;
      _w7 : Bool;
      _w8 : Bool;
      _w9 : Bool;
      _w10 : Bool;
      _w11 : Bool;
      _w12 : Bool;
      _w13 : Bool;
      _w14 : Bool;
      _w15 : Bool;
      _w16 : Bool;
   END_VAR
BEGIN

REGION Network 1: Устройство в ручном режиме
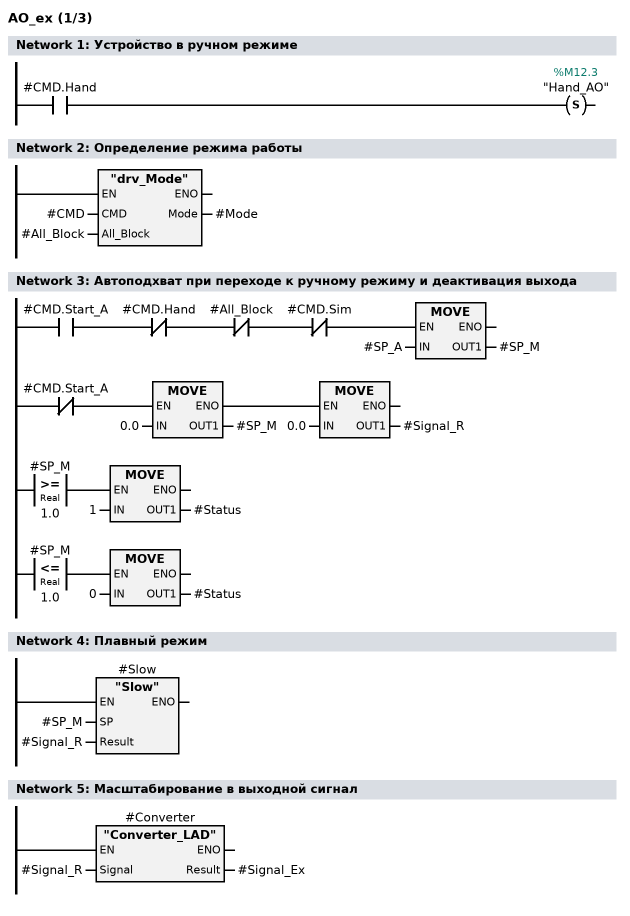
   RUNG wire#powerrail
      Contact( #CMD.Hand )
      S_Coil( "Hand_AO" )
   END_RUNG
   // the same network as SCL:
   IF #CMD.Hand THEN "Hand_AO" := TRUE; END_IF;
END_REGION

REGION Network 2: Определение режима работы
   RUNG wire#powerrail
      "drv_Mode"(CMD := #CMD, All_Block := #All_Block, Mode => #Mode)
   END_RUNG
   // the same network as SCL:
   "drv_Mode"(CMD := #CMD, All_Block := #All_Block, Mode => #Mode);
END_REGION

REGION Network 3: Автоподхват при переходе к ручному режиму и деактивация выхода
   RUNG wire#powerrail
      Contact( #CMD.Start_A )
      I_Contact( #CMD.Hand )
      I_Contact( #All_Block )
      I_Contact( #CMD.Sim )
      { S7_GenerateENO := "TRUE" } Move(in := #SP_A, out1 => #SP_M)
   END_RUNG
   RUNG wire#powerrail
      I_Contact( #CMD.Start_A )
      { S7_GenerateENO := "TRUE" } Move(in := 0.0, out1 => #SP_M)
      { S7_GenerateENO := "TRUE" } Move(in := 0.0, out1 => #Signal_R)
   END_RUNG
   RUNG wire#powerrail
      { S7_Templates := "SrcType := Real" } GE_Contact(in1 := #SP_M, in2 := 1.0)
      Move(in := 1, out1 => #Status)
   END_RUNG
   RUNG wire#powerrail
      { S7_Templates := "SrcType := Real" } LE_Contact(in1 := #SP_M, in2 := 1.0)
      Move(in := 0, out1 => #Status)
   END_RUNG
   // the same network as SCL:
   // ENO of a box is taken as its EN; it also drops when the box reports an error
   IF #CMD.Start_A AND NOT #CMD.Hand AND NOT #All_Block AND NOT #CMD.Sim THEN #SP_M := #SP_A; END_IF;
   IF NOT #CMD.Start_A THEN
       #SP_M := 0.0;
       #Signal_R := 0.0;
   END_IF;
   IF #SP_M >= 1.0 THEN #Status := 1; END_IF;
   IF #SP_M <= 1.0 THEN #Status := 0; END_IF;
END_REGION

REGION Network 4: Плавный режим
   RUNG wire#powerrail
      #Slow(SP := #SP_M, Result := #Signal_R)
   END_RUNG
   // the same network as SCL:
   #Slow(SP := #SP_M, Result := #Signal_R);   // "Slow"
END_REGION

REGION Network 5: Масштабирование в выходной сигнал
   RUNG wire#powerrail
      #Converter(Signal := #Signal_R, Result => #Signal_Ex)
   END_RUNG
   // the same network as SCL:
   #Converter(Signal := #Signal_R, Result => #Signal_Ex);   // "Converter_LAD"
END_REGION

REGION Network 6: Преобразование кода в реальное значение входа
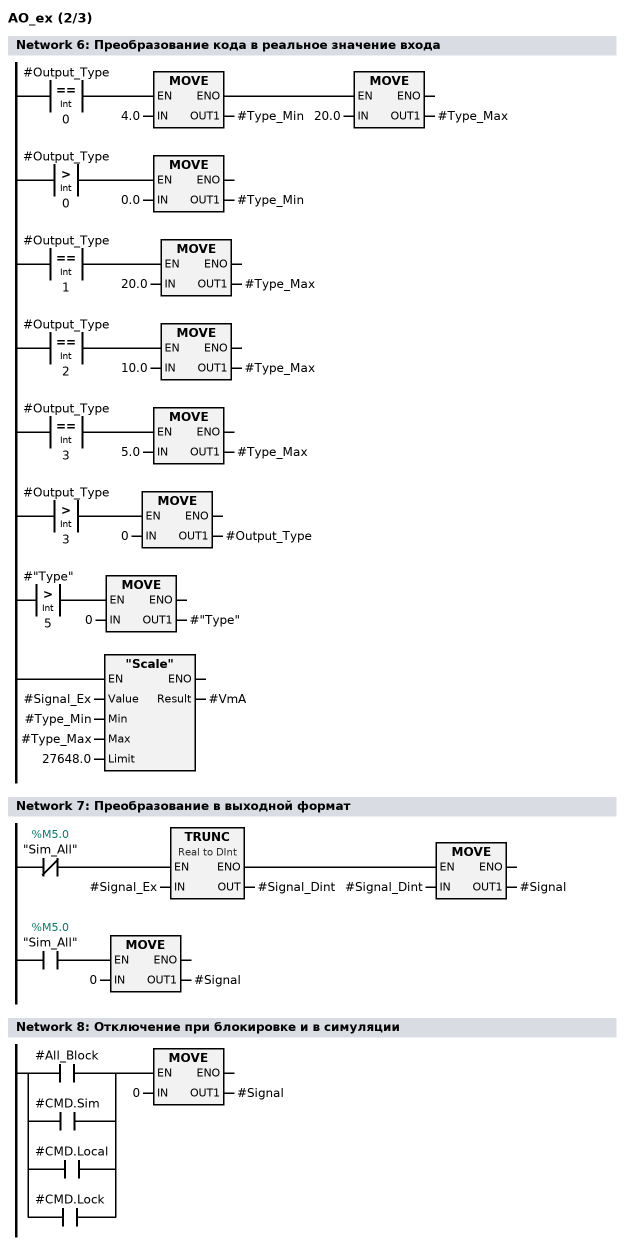
   RUNG wire#powerrail
      { S7_Templates := "SrcType := Int" } EQ_Contact(in1 := #Output_Type, in2 := 0)
      Move(in := 4.0, out1 => #Type_Min)
      Move(in := 20.0, out1 => #Type_Max)
   END_RUNG
   RUNG wire#powerrail
      { S7_Templates := "SrcType := Int" } GT_Contact(in1 := #Output_Type, in2 := 0)
      Move(in := 0.0, out1 => #Type_Min)
   END_RUNG
   RUNG wire#powerrail
      { S7_Templates := "SrcType := Int" } EQ_Contact(in1 := #Output_Type, in2 := 1)
      Move(in := 20.0, out1 => #Type_Max)
   END_RUNG
   RUNG wire#powerrail
      { S7_Templates := "SrcType := Int" } EQ_Contact(in1 := #Output_Type, in2 := 2)
      Move(in := 10.0, out1 => #Type_Max)
   END_RUNG
   RUNG wire#powerrail
      { S7_Templates := "SrcType := Int" } EQ_Contact(in1 := #Output_Type, in2 := 3)
      Move(in := 5.0, out1 => #Type_Max)
   END_RUNG
   RUNG wire#powerrail
      { S7_Templates := "SrcType := Int" } GT_Contact(in1 := #Output_Type, in2 := 3)
      Move(in := 0, out1 => #Output_Type)
   END_RUNG
   RUNG wire#powerrail
      { S7_Templates := "SrcType := Int" } GT_Contact(in1 := #"Type", in2 := 5)
      Move(in := 0, out1 => #"Type")
   END_RUNG
   RUNG wire#powerrail
      "Scale"(Value := #Signal_Ex, Min := #Type_Min, Max := #Type_Max, Limit := 27648.0, Result => #VmA)
   END_RUNG
   // the same network as SCL:
   IF #Output_Type = 0 THEN
       #Type_Min := 4.0;
       #Type_Max := 20.0;
   END_IF;
   IF #Output_Type > 0 THEN #Type_Min := 0.0; END_IF;
   IF #Output_Type = 1 THEN #Type_Max := 20.0; END_IF;
   IF #Output_Type = 2 THEN #Type_Max := 10.0; END_IF;
   IF #Output_Type = 3 THEN #Type_Max := 5.0; END_IF;
   IF #Output_Type > 3 THEN #Output_Type := 0; END_IF;
   IF #"Type" > 5 THEN #"Type" := 0; END_IF;
   "Scale"(Value := #Signal_Ex, Min := #Type_Min, Max := #Type_Max, Limit := 27648.0, Result => #VmA);
END_REGION

REGION Network 7: Преобразование в выходной формат
   RUNG wire#powerrail
      I_Contact( "Sim_All" )
      { S7_Templates := "[SrcType := Real, DestType := DInt]"; S7_GenerateENO := "TRUE" } Trunc(in := #Signal_Ex, out => #Signal_Dint)
      { S7_GenerateENO := "TRUE" } Move(in := #Signal_Dint, out1 => #Signal)
   END_RUNG
   RUNG wire#powerrail
      Contact( "Sim_All" )
      { S7_GenerateENO := "TRUE" } Move(in := 0, out1 => #Signal)
   END_RUNG
   // the same network as SCL:
   // ENO of a box is taken as its EN; it also drops when the box reports an error
   IF NOT "Sim_All" THEN
       #Signal_Dint := TRUNC(#Signal_Ex);
       #Signal := #Signal_Dint;
   END_IF;
   IF "Sim_All" THEN #Signal := 0; END_IF;
END_REGION

REGION Network 8: Отключение при блокировке и в симуляции
   RUNG wire#powerrail
      Contact( #All_Block )
      wire#w1
      { S7_GenerateENO := "TRUE" } Move(in := 0, out1 => #Signal)
   END_RUNG
   RUNG wire#powerrail
      Contact( #CMD.Sim )
   END_RUNG wire#w1
   RUNG wire#powerrail
      Contact( #CMD.Local )
   END_RUNG wire#w1
   RUNG wire#powerrail
      Contact( #CMD.Lock )
   END_RUNG wire#w1
   // the same network as SCL:
   IF #All_Block OR #CMD.Sim OR #CMD.Local OR #CMD.Lock THEN #Signal := 0; END_IF;
END_REGION

REGION Network 9: События выхода
   // 0 - выход активирован
   // 1 - выход деактивирован
   // 2 - выход в ручном режиме
   // 3 - выход в автоматическом режиме
   // 4 - плавный разгон активирован
   // 5 - плавный разгон деактивирован
   // 6 - плавное замедление активировано
   // 7 - плавное замедление деактивировано
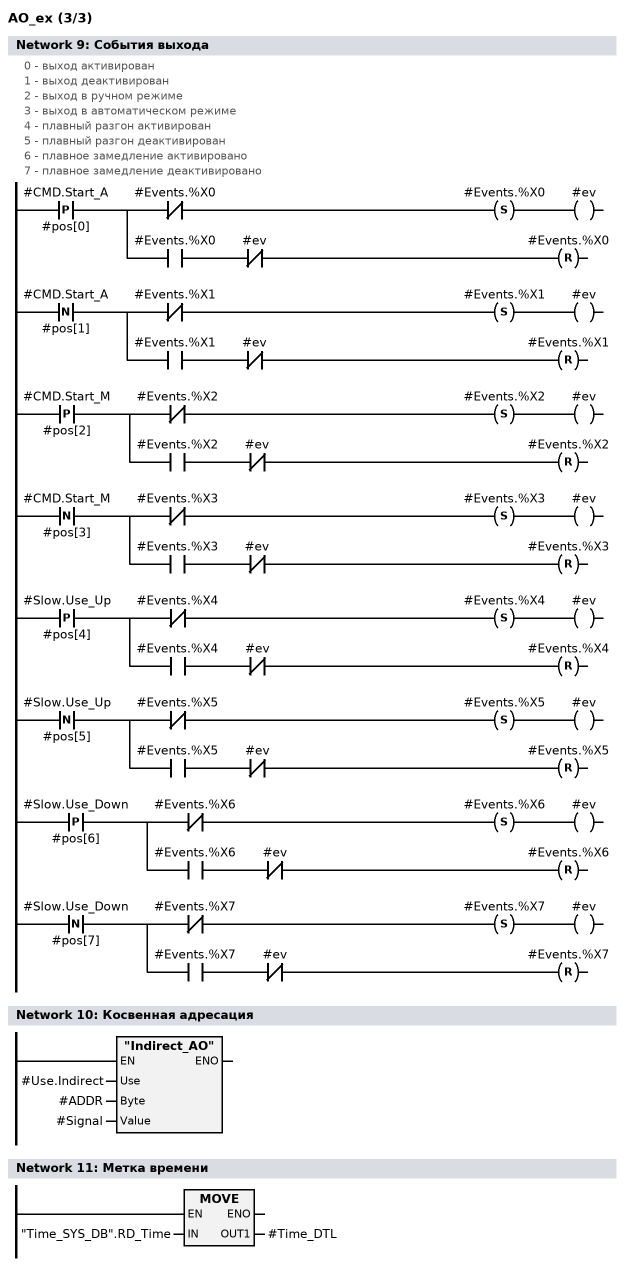
   RUNG wire#powerrail
      P_Contact(operand := #CMD.Start_A, bit := #pos[0])
      wire#w1
      I_Contact( #Events.%X0 )
      S_Coil( #Events.%X0 )
      Coil( #ev )
   END_RUNG
   RUNG wire#w1
      Contact( #Events.%X0 )
      I_Contact( #ev )
      R_Coil( #Events.%X0 )
   END_RUNG
   RUNG wire#powerrail
      N_Contact(operand := #CMD.Start_A, bit := #pos[1])
      wire#w2
      I_Contact( #Events.%X1 )
      S_Coil( #Events.%X1 )
      Coil( #ev )
   END_RUNG
   RUNG wire#w2
      Contact( #Events.%X1 )
      I_Contact( #ev )
      R_Coil( #Events.%X1 )
   END_RUNG
   RUNG wire#powerrail
      P_Contact(operand := #CMD.Start_M, bit := #pos[2])
      wire#w3
      I_Contact( #Events.%X2 )
      S_Coil( #Events.%X2 )
      Coil( #ev )
   END_RUNG
   RUNG wire#w3
      Contact( #Events.%X2 )
      I_Contact( #ev )
      R_Coil( #Events.%X2 )
   END_RUNG
   RUNG wire#powerrail
      N_Contact(operand := #CMD.Start_M, bit := #pos[3])
      wire#w4
      I_Contact( #Events.%X3 )
      S_Coil( #Events.%X3 )
      Coil( #ev )
   END_RUNG
   RUNG wire#w4
      Contact( #Events.%X3 )
      I_Contact( #ev )
      R_Coil( #Events.%X3 )
   END_RUNG
   RUNG wire#powerrail
      P_Contact(operand := #Slow.Use_Up, bit := #pos[4])
      wire#w5
      I_Contact( #Events.%X4 )
      S_Coil( #Events.%X4 )
      Coil( #ev )
   END_RUNG
   RUNG wire#w5
      Contact( #Events.%X4 )
      I_Contact( #ev )
      R_Coil( #Events.%X4 )
   END_RUNG
   RUNG wire#powerrail
      N_Contact(operand := #Slow.Use_Up, bit := #pos[5])
      wire#w6
      I_Contact( #Events.%X5 )
      S_Coil( #Events.%X5 )
      Coil( #ev )
   END_RUNG
   RUNG wire#w6
      Contact( #Events.%X5 )
      I_Contact( #ev )
      R_Coil( #Events.%X5 )
   END_RUNG
   RUNG wire#powerrail
      P_Contact(operand := #Slow.Use_Down, bit := #pos[6])
      wire#w7
      I_Contact( #Events.%X6 )
      S_Coil( #Events.%X6 )
      Coil( #ev )
   END_RUNG
   RUNG wire#w7
      Contact( #Events.%X6 )
      I_Contact( #ev )
      R_Coil( #Events.%X6 )
   END_RUNG
   RUNG wire#powerrail
      N_Contact(operand := #Slow.Use_Down, bit := #pos[7])
      wire#w8
      I_Contact( #Events.%X7 )
      S_Coil( #Events.%X7 )
      Coil( #ev )
   END_RUNG
   RUNG wire#w8
      Contact( #Events.%X7 )
      I_Contact( #ev )
      R_Coil( #Events.%X7 )
   END_RUNG
   // the same network as SCL:
   #_w1 := #CMD.Start_A AND NOT #pos[0];   // rising edge of #CMD.Start_A
   #pos[0] := #CMD.Start_A;
   #_w2 := #_w1 AND NOT #Events.%X0;
   IF #_w2 THEN #Events.%X0 := TRUE; END_IF;
   #ev := #_w2;
   IF #_w1 AND #Events.%X0 AND NOT #ev THEN #Events.%X0 := FALSE; END_IF;
   #_w3 := NOT #CMD.Start_A AND #pos[1];   // falling edge of #CMD.Start_A
   #pos[1] := #CMD.Start_A;
   #_w4 := #_w3 AND NOT #Events.%X1;
   IF #_w4 THEN #Events.%X1 := TRUE; END_IF;
   #ev := #_w4;
   IF #_w3 AND #Events.%X1 AND NOT #ev THEN #Events.%X1 := FALSE; END_IF;
   #_w5 := #CMD.Start_M AND NOT #pos[2];   // rising edge of #CMD.Start_M
   #pos[2] := #CMD.Start_M;
   #_w6 := #_w5 AND NOT #Events.%X2;
   IF #_w6 THEN #Events.%X2 := TRUE; END_IF;
   #ev := #_w6;
   IF #_w5 AND #Events.%X2 AND NOT #ev THEN #Events.%X2 := FALSE; END_IF;
   #_w7 := NOT #CMD.Start_M AND #pos[3];   // falling edge of #CMD.Start_M
   #pos[3] := #CMD.Start_M;
   #_w8 := #_w7 AND NOT #Events.%X3;
   IF #_w8 THEN #Events.%X3 := TRUE; END_IF;
   #ev := #_w8;
   IF #_w7 AND #Events.%X3 AND NOT #ev THEN #Events.%X3 := FALSE; END_IF;
   #_w9 := #Slow.Use_Up AND NOT #pos[4];   // rising edge of #Slow.Use_Up
   #pos[4] := #Slow.Use_Up;
   #_w10 := #_w9 AND NOT #Events.%X4;
   IF #_w10 THEN #Events.%X4 := TRUE; END_IF;
   #ev := #_w10;
   IF #_w9 AND #Events.%X4 AND NOT #ev THEN #Events.%X4 := FALSE; END_IF;
   #_w11 := NOT #Slow.Use_Up AND #pos[5];   // falling edge of #Slow.Use_Up
   #pos[5] := #Slow.Use_Up;
   #_w12 := #_w11 AND NOT #Events.%X5;
   IF #_w12 THEN #Events.%X5 := TRUE; END_IF;
   #ev := #_w12;
   IF #_w11 AND #Events.%X5 AND NOT #ev THEN #Events.%X5 := FALSE; END_IF;
   #_w13 := #Slow.Use_Down AND NOT #pos[6];   // rising edge of #Slow.Use_Down
   #pos[6] := #Slow.Use_Down;
   #_w14 := #_w13 AND NOT #Events.%X6;
   IF #_w14 THEN #Events.%X6 := TRUE; END_IF;
   #ev := #_w14;
   IF #_w13 AND #Events.%X6 AND NOT #ev THEN #Events.%X6 := FALSE; END_IF;
   #_w15 := NOT #Slow.Use_Down AND #pos[7];   // falling edge of #Slow.Use_Down
   #pos[7] := #Slow.Use_Down;
   #_w16 := #_w15 AND NOT #Events.%X7;
   IF #_w16 THEN #Events.%X7 := TRUE; END_IF;
   #ev := #_w16;
   IF #_w15 AND #Events.%X7 AND NOT #ev THEN #Events.%X7 := FALSE; END_IF;
END_REGION

REGION Network 10: Косвенная адресация
   RUNG wire#powerrail
      "Indirect_AO"(Use := #Use.Indirect, "Byte" := #ADDR, Value := #Signal)
   END_RUNG
   // the same network as SCL:
   "Indirect_AO"(Use := #Use.Indirect, "Byte" := #ADDR, Value := #Signal);
END_REGION

REGION Network 11: Метка времени
   RUNG wire#powerrail
      Move(in := "Time_SYS_DB".RD_Time, out1 => #Time_DTL)
   END_RUNG
   // the same network as SCL:
   #Time_DTL := "Time_SYS_DB".RD_Time;
END_REGION
END_FUNCTION_BLOCK

FUNCTION_BLOCK "Slow"   // FB151, LAD
{ S7_Optimized_Access := 'FALSE' }
VERSION : 0.1
// stored: AutoNumber false, IsIECCheckEnabled false, SetENOAutomatically false, UDAEnableTagReadback false
   VAR_INPUT
      SP : Real;   // Уставка
   END_VAR
   VAR_IN_OUT
      Result : Real;   // Управляющий сигнал
   END_VAR
   VAR DB_SPECIFIC
      Use_Up { S7_SetPoint := 'True'} : Bool;   // Использовать плавный разгон
      Use_Down { S7_SetPoint := 'True'} : Bool;   // Использовать плавное замедление
      Active : Bool;   // Идёт изменение уставки
      Active_Up : Bool;
      Active_Down : Bool;
      Step_Up { S7_SetPoint := 'True'} : Real := 0.125;   // Шаг плавного разгона
      Step_Down { S7_SetPoint := 'True'} : Real := 0.125;   // Шаг плавного замедления
   END_VAR
   VAR
      T_Up { S7_SetPoint := 'True'} : "Time_R";   // Таймер плавного разгона
      T_Down { S7_SetPoint := 'True'} : "Time_R";   // Таймер плавного замедления
   END_VAR
   VAR_TEMP
      Delta_Up : Real;   // Отклонение сигнала от уставки
      Delta_Down : Real;
   END_VAR
   VAR_TEMP   // added for the SCL form of the ladder/FBD networks
      _w1 : Bool;
      _w2 : Bool;
   END_VAR
BEGIN

REGION Network 1: Не используется
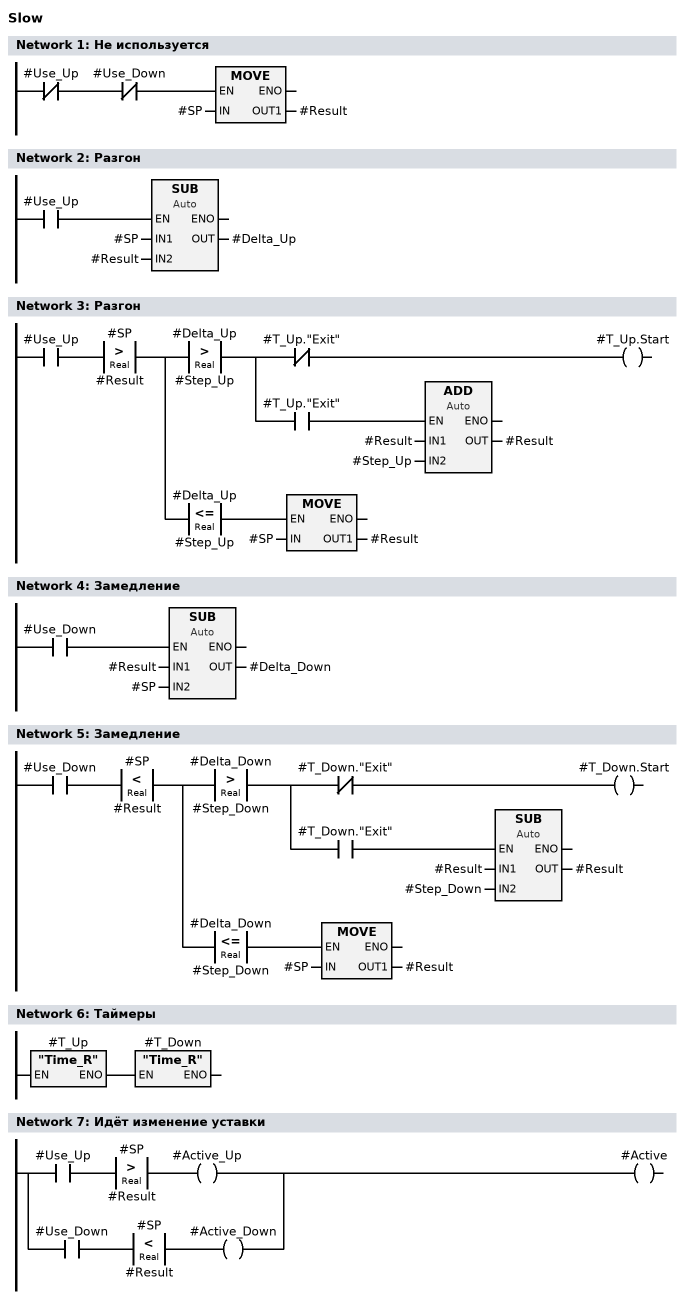
   RUNG wire#powerrail
      I_Contact( #Use_Up )
      I_Contact( #Use_Down )
      Move(in := #SP, out1 => #Result)
   END_RUNG
   // the same network as SCL:
   IF NOT #Use_Up AND NOT #Use_Down THEN #Result := #SP; END_IF;
END_REGION

REGION Network 2: Разгон
   RUNG wire#powerrail
      Contact( #Use_Up )
      Sub(in1 := #SP, in2 := #Result, out => #Delta_Up)
   END_RUNG
   // the same network as SCL:
   IF #Use_Up THEN #Delta_Up := #SP - #Result; END_IF;
END_REGION

REGION Network 3: Разгон
   RUNG wire#powerrail
      Contact( #Use_Up )
      { S7_Templates := "SrcType := Real" } GT_Contact(in1 := #SP, in2 := #Result)
      wire#w1
      { S7_Templates := "SrcType := Real" } GT_Contact(in1 := #Delta_Up, in2 := #Step_Up)
      wire#w2
      I_Contact( #T_Up."Exit" )
      Coil( #T_Up.Start )
   END_RUNG
   RUNG wire#w2
      Contact( #T_Up."Exit" )
      Add(in1 := #Result, in2 := #Step_Up, out => #Result)
   END_RUNG
   RUNG wire#w1
      { S7_Templates := "SrcType := Real" } LE_Contact(in1 := #Delta_Up, in2 := #Step_Up)
      Move(in := #SP, out1 => #Result)
   END_RUNG
   // the same network as SCL:
   #_w1 := #Use_Up AND (#SP > #Result);
   #_w2 := #_w1 AND (#Delta_Up > #Step_Up);
   #T_Up.Start := #_w2 AND NOT #T_Up."Exit";
   IF #_w2 AND #T_Up."Exit" THEN #Result := #Result + #Step_Up; END_IF;
   IF #_w1 AND (#Delta_Up <= #Step_Up) THEN #Result := #SP; END_IF;
END_REGION

REGION Network 4: Замедление
   RUNG wire#powerrail
      Contact( #Use_Down )
      Sub(in1 := #Result, in2 := #SP, out => #Delta_Down)
   END_RUNG
   // the same network as SCL:
   IF #Use_Down THEN #Delta_Down := #Result - #SP; END_IF;
END_REGION

REGION Network 5: Замедление
   RUNG wire#powerrail
      Contact( #Use_Down )
      { S7_Templates := "SrcType := Real" } LT_Contact(in1 := #SP, in2 := #Result)
      wire#w1
      { S7_Templates := "SrcType := Real" } GT_Contact(in1 := #Delta_Down, in2 := #Step_Down)
      wire#w2
      I_Contact( #T_Down."Exit" )
      Coil( #T_Down.Start )
   END_RUNG
   RUNG wire#w2
      Contact( #T_Down."Exit" )
      Sub(in1 := #Result, in2 := #Step_Down, out => #Result)
   END_RUNG
   RUNG wire#w1
      { S7_Templates := "SrcType := Real" } LE_Contact(in1 := #Delta_Down, in2 := #Step_Down)
      Move(in := #SP, out1 => #Result)
   END_RUNG
   // the same network as SCL:
   #_w1 := #Use_Down AND (#SP < #Result);
   #_w2 := #_w1 AND (#Delta_Down > #Step_Down);
   #T_Down.Start := #_w2 AND NOT #T_Down."Exit";
   IF #_w2 AND #T_Down."Exit" THEN #Result := #Result - #Step_Down; END_IF;
   IF #_w1 AND (#Delta_Down <= #Step_Down) THEN #Result := #SP; END_IF;
END_REGION

REGION Network 6: Таймеры
   RUNG wire#powerrail
      #T_Up()
      #T_Down()
   END_RUNG
   // the same network as SCL:
   #T_Up(ENO => #_w1);   // "Time_R"
   IF #_w1 THEN
       #T_Down();   // "Time_R"
   END_IF;
END_REGION

REGION Network 7: Идёт изменение уставки
   RUNG wire#powerrail
      Contact( #Use_Up )
      { S7_Templates := "SrcType := Real" } GT_Contact(in1 := #SP, in2 := #Result)
      Coil( #Active_Up )
      wire#w1
      Coil( #Active )
   END_RUNG
   RUNG wire#powerrail
      Contact( #Use_Down )
      { S7_Templates := "SrcType := Real" } LT_Contact(in1 := #SP, in2 := #Result)
      Coil( #Active_Down )
   END_RUNG wire#w1
   // the same network as SCL:
   #Active_Up := #Use_Up AND (#SP > #Result);
   #Active_Down := #Use_Down AND (#SP < #Result);
   #Active := #Active_Up OR #Active_Down;
END_REGION
END_FUNCTION_BLOCK

FUNCTION_BLOCK "Motors"   // FB240, LAD
{ S7_Optimized_Access := 'FALSE' }
VERSION : 0.1
// stored: AutoNumber false, IsIECCheckEnabled false, SetENOAutomatically false, UDAEnableTagReadback false
   VAR DB_SPECIFIC
      Time_DTL { S7_SetPoint := 'True'} : DTL;
   END_VAR
   VAR_TEMP   // added for the SCL form of the ladder/FBD networks
      _w1 : Bool;
   END_VAR
BEGIN

REGION Network 1: Мешалки
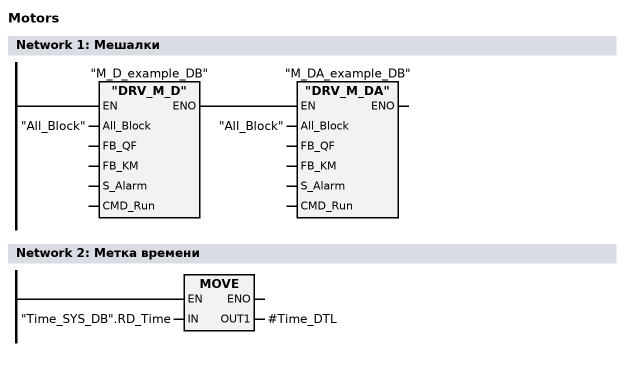
   RUNG wire#powerrail
      "M_D_example_DB"(All_Block := "All_Block", FB_QF :=, FB_KM :=, S_Alarm :=, CMD_Run :=)
      "M_DA_example_DB"(All_Block := "All_Block", FB_QF :=, FB_KM :=, S_Alarm :=, CMD_Run :=)
   END_RUNG
   // the same network as SCL:
   "M_D_example_DB"(All_Block := "All_Block", ENO => #_w1);   // "DRV_M_D"
   IF #_w1 THEN
       "M_DA_example_DB"(All_Block := "All_Block");   // "DRV_M_DA"
   END_IF;
END_REGION

REGION Network 2: Метка времени
   RUNG wire#powerrail
      Move(in := "Time_SYS_DB".RD_Time, out1 => #Time_DTL)
   END_RUNG
   // the same network as SCL:
   #Time_DTL := "Time_SYS_DB".RD_Time;
END_REGION
END_FUNCTION_BLOCK

FUNCTION_BLOCK "DRV_M_D"   // FB110, LAD
{ S7_Optimized_Access := 'FALSE' }
VERSION : 0.1
// stored: AutoNumber false, IsIECCheckEnabled false, SetENOAutomatically false, UDAEnableTagReadback false
   VAR_INPUT
      All_Block : Bool;   // Аварийный останов
   END_VAR
   VAR_IN_OUT
      FB_QF : Bool;   // защитный автомат / Защитный автомат / Готовность
      FB_KM : Bool;   // привод запущен / Пускатель / В работе
      S_Alarm : Bool;   // Внешний индикатор наличия аварии
      CMD_Run : Bool;   // Команда запуска двигателя
   END_VAR
   VAR DB_SPECIFIC
      CMD : "CMD";   // Основные команды / Блок команд
      Mode : Int;   // Режим работы
      Status : Int;   // Статус устройства
      Use : Struct   // Функционал
         QF { S7_SetPoint := 'True'} : Bool := true;   // Защитный автомат
         KM { S7_SetPoint := 'True'} : Bool := true;   // Пускатель
         OpTime { S7_SetPoint := 'True'} : Bool := true;   // Контроль наработки
         Analog { S7_SetPoint := 'True'} : Bool;
         Local_Keys : Bool;
      END_STRUCT;
      FB : Struct   // Функционал
         QF : Bool;   // Защитный автомат
         KM : Bool;   // Пускатель
         Local_Start : Bool;
         Local_Stop : Bool;
      END_STRUCT;
      ON : Bool;   // Успешно запущено
      OFF : Bool;   // Успешно остановлено
   END_VAR
   VAR
      Tx { S7_SetPoint := 'True'} : Array[0..3] of "Time_S";   // Блок таймеров
   END_VAR
   VAR DB_SPECIFIC
      Inv : Struct   // Инверсия сигналов
         CMD { S7_SetPoint := 'True'} : Bool;   // Команда запуска
         QF { S7_SetPoint := 'True'} : Bool;   // Защитный автомат
         KM { S7_SetPoint := 'True'} : Bool;   // Пускатель
      END_STRUCT;
      Alarm : Struct   // Сбор аварий / Список аварий
         Block : Bool;   // Аварийная остановка
         QF : Bool;   // привод не готов / Выбило защитный автомат
         Start : Bool;   // Ошибка при запуске
         Stop : Bool;   // Ошибка при останове
         Termo : Bool;   // термозащита / Сработала термозащита
         Alarm : Bool;   // Внешняя авария
         Safety : Bool;   // Сработала безопасность
         OpTime : Bool;
      END_STRUCT;
      Alarms : Word;   // Слово аварий
      Events : Word;   // События
      pos : Array[0..15] of Bool;
      OpTime_h : DInt;   // наработка (ч)
      OpTime_s { S7_SetPoint := 'True'} : DInt;   // наработка (с)
      OpTime_SP { S7_SetPoint := 'True'} : DInt := 2160;   // Интервал обслуживания, ч
      OpTime_Now_h : DInt;   // Прошло с прошлого обслуживания, ч
      OpTime_Now_s { S7_SetPoint := 'True'} : DInt;   // Прошло с прошлого обслуживания, с
      CodeID { S7_SetPoint := 'True'} : Int;   // Код датчика для привязки в скаде
      Indirect : Struct   // Использование косвенной адресации
         FB_QF { S7_SetPoint := 'True'} : Bool := true;   // Защитный автомат
         FB_KM { S7_SetPoint := 'True'} : Bool := true;   // Пускатель
         CMD { S7_SetPoint := 'True'} : Bool := true;   // Запуск двигателя
      END_STRUCT;
      Indirect_BYTE : Struct   // Адрес входа на контроллере (Байт)
         FB_QF { S7_SetPoint := 'True'} : Int;   // Защитный автомат
         FB_KM { S7_SetPoint := 'True'} : Int;   // Пускатель
         CMD { S7_SetPoint := 'True'} : Int;   // Запуск двигателя
      END_STRUCT;
      Indirect_BIT : Struct   // Адрес входа на контроллере (Бит)
         FB_QF { S7_SetPoint := 'True'} : Int := 9;   // Защитный автомат
         FB_KM { S7_SetPoint := 'True'} : Int := 9;   // Пускатель
         CMD { S7_SetPoint := 'True'} : Int := 9;   // Запуск двигателя
      END_STRUCT;
      Time_DTL : DTL;
   END_VAR
   VAR_TEMP
      ev : Bool;
      xQF : Bool;
      xKM : Bool;
   END_VAR
   VAR_TEMP   // added for the SCL form of the ladder/FBD networks
      _w1 : Bool;
      _w2 : Bool;
      _w3 : Bool;
      _w4 : Bool;
      _w5 : Bool;
      _w6 : Bool;
      _w7 : Bool;
      _w8 : Bool;
      _w9 : Bool;
      _w10 : Bool;
      _w11 : Bool;
      _w12 : Bool;
      _w13 : Bool;
      _w14 : Bool;
      _w15 : Bool;
      _w16 : Bool;
      _w17 : Bool;
      _w18 : Bool;
      _w19 : Bool;
      _w20 : Bool;
      _w21 : Bool;
      _w22 : Bool;
      _w23 : Bool;
      _w24 : Bool;
      _w25 : Bool;
      _w26 : Bool;
   END_VAR
BEGIN

REGION Network 1: Режим глобальной симуляции
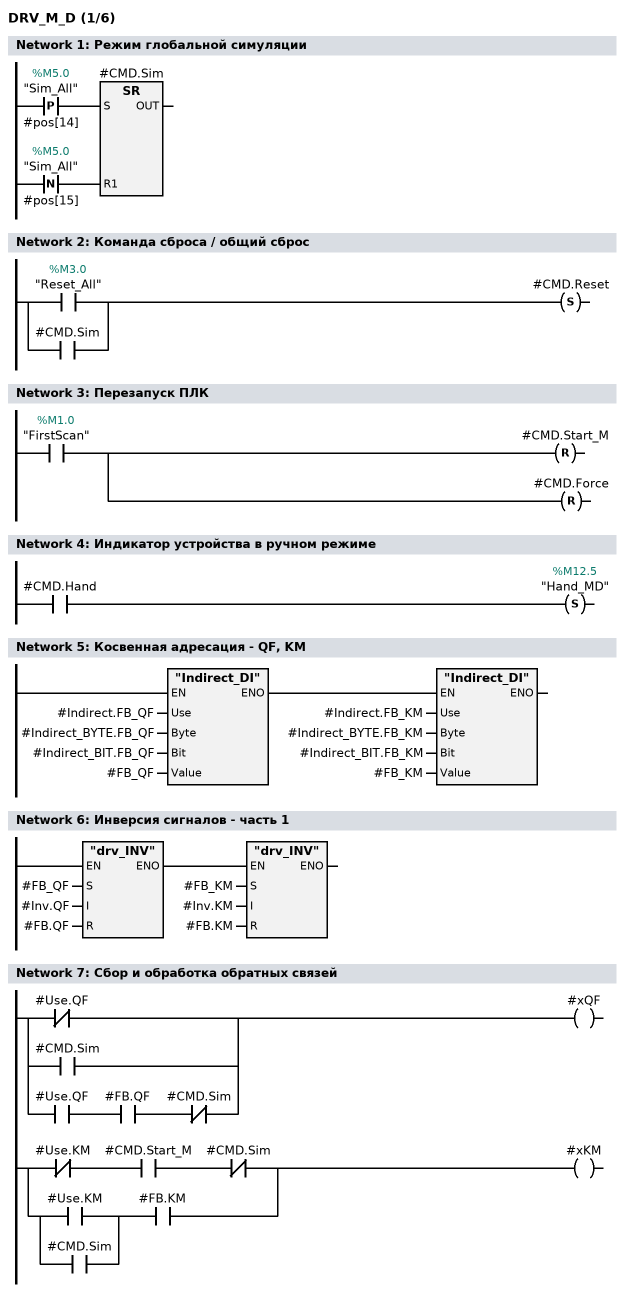
   RUNG wire#powerrail
      P_Contact(operand := "Sim_All", bit := #pos[14])
      S_SR(operand := #CMD.Sim, r1 := wire#w1)
   END_RUNG
   RUNG wire#powerrail
      N_Contact(operand := "Sim_All", bit := #pos[15])
   END_RUNG wire#w1
   // the same network as SCL:
   #_w1 := "Sim_All" AND NOT #pos[14];   // rising edge of "Sim_All"
   #pos[14] := "Sim_All";
   #_w2 := NOT "Sim_All" AND #pos[15];   // falling edge of "Sim_All"
   #pos[15] := "Sim_All";
   IF #_w1 THEN
       #CMD.Sim := TRUE;   // SR flip-flop
   END_IF;
   IF #_w2 THEN #CMD.Sim := FALSE; END_IF;
END_REGION

REGION Network 2: Команда сброса / общий сброс
   RUNG wire#powerrail
      Contact( "Reset_All" )
      wire#w1
      S_Coil( #CMD.Reset )
   END_RUNG
   RUNG wire#powerrail
      Contact( #CMD.Sim )
   END_RUNG wire#w1
   // the same network as SCL:
   IF "Reset_All" OR #CMD.Sim THEN #CMD.Reset := TRUE; END_IF;
END_REGION

REGION Network 3: Перезапуск ПЛК
   RUNG wire#powerrail
      Contact( "FirstScan" )
      wire#w1
      R_Coil( #CMD.Start_M )
   END_RUNG
   RUNG wire#w1
      R_Coil( #CMD.Force )
   END_RUNG
   // the same network as SCL:
   IF "FirstScan" THEN
       #CMD.Start_M := FALSE;
       #CMD.Force := FALSE;
   END_IF;
END_REGION

REGION Network 4: Индикатор устройства в ручном режиме
   RUNG wire#powerrail
      Contact( #CMD.Hand )
      S_Coil( "Hand_MD" )
   END_RUNG
   // the same network as SCL:
   IF #CMD.Hand THEN "Hand_MD" := TRUE; END_IF;
END_REGION

REGION Network 5: Косвенная адресация - QF, KM
   RUNG wire#powerrail
      "Indirect_DI"(Use := #Indirect.FB_QF, "Byte" := #Indirect_BYTE.FB_QF, Bit := #Indirect_BIT.FB_QF, Value := #FB_QF)
      "Indirect_DI"(Use := #Indirect.FB_KM, "Byte" := #Indirect_BYTE.FB_KM, Bit := #Indirect_BIT.FB_KM, Value := #FB_KM)
   END_RUNG
   // the same network as SCL:
   "Indirect_DI"(Use := #Indirect.FB_QF,
                 "Byte" := #Indirect_BYTE.FB_QF,
                 Bit := #Indirect_BIT.FB_QF,
                 Value := #FB_QF,
                 ENO => #_w1);
   IF #_w1 THEN
       "Indirect_DI"(Use := #Indirect.FB_KM,
                     "Byte" := #Indirect_BYTE.FB_KM,
                     Bit := #Indirect_BIT.FB_KM,
                     Value := #FB_KM);
   END_IF;
END_REGION

REGION Network 6: Инверсия сигналов - часть 1
   RUNG wire#powerrail
      "drv_INV"(S := #FB_QF, I := #Inv.QF, R := #FB.QF)
      "drv_INV"(S := #FB_KM, I := #Inv.KM, R := #FB.KM)
   END_RUNG
   // the same network as SCL:
   "drv_INV"(S := #FB_QF, I := #Inv.QF, R := #FB.QF, ENO => #_w1);
   IF #_w1 THEN "drv_INV"(S := #FB_KM, I := #Inv.KM, R := #FB.KM); END_IF;
END_REGION

REGION Network 7: Сбор и обработка обратных связей
   RUNG wire#powerrail
      I_Contact( #Use.QF )
      wire#w1
      Coil( #xQF )
   END_RUNG
   RUNG wire#powerrail
      Contact( #CMD.Sim )
   END_RUNG wire#w1
   RUNG wire#powerrail
      Contact( #Use.QF )
      Contact( #FB.QF )
      I_Contact( #CMD.Sim )
   END_RUNG wire#w1
   RUNG wire#powerrail
      I_Contact( #Use.KM )
      Contact( #CMD.Start_M )
      I_Contact( #CMD.Sim )
      wire#w2
      Coil( #xKM )
   END_RUNG
   RUNG wire#powerrail
      Contact( #Use.KM )
      wire#w3
      Contact( #FB.KM )
   END_RUNG wire#w2
   RUNG wire#powerrail
      Contact( #CMD.Sim )
   END_RUNG wire#w3
   // the same network as SCL:
   #xQF := NOT #Use.QF OR #CMD.Sim OR (#Use.QF AND #FB.QF AND NOT #CMD.Sim);
   #xKM := (NOT #Use.KM AND #CMD.Start_M AND NOT #CMD.Sim) OR ((#Use.KM OR #CMD.Sim) AND #FB.KM);
END_REGION

REGION Network 8: Режим работы устройства / определение режима работы
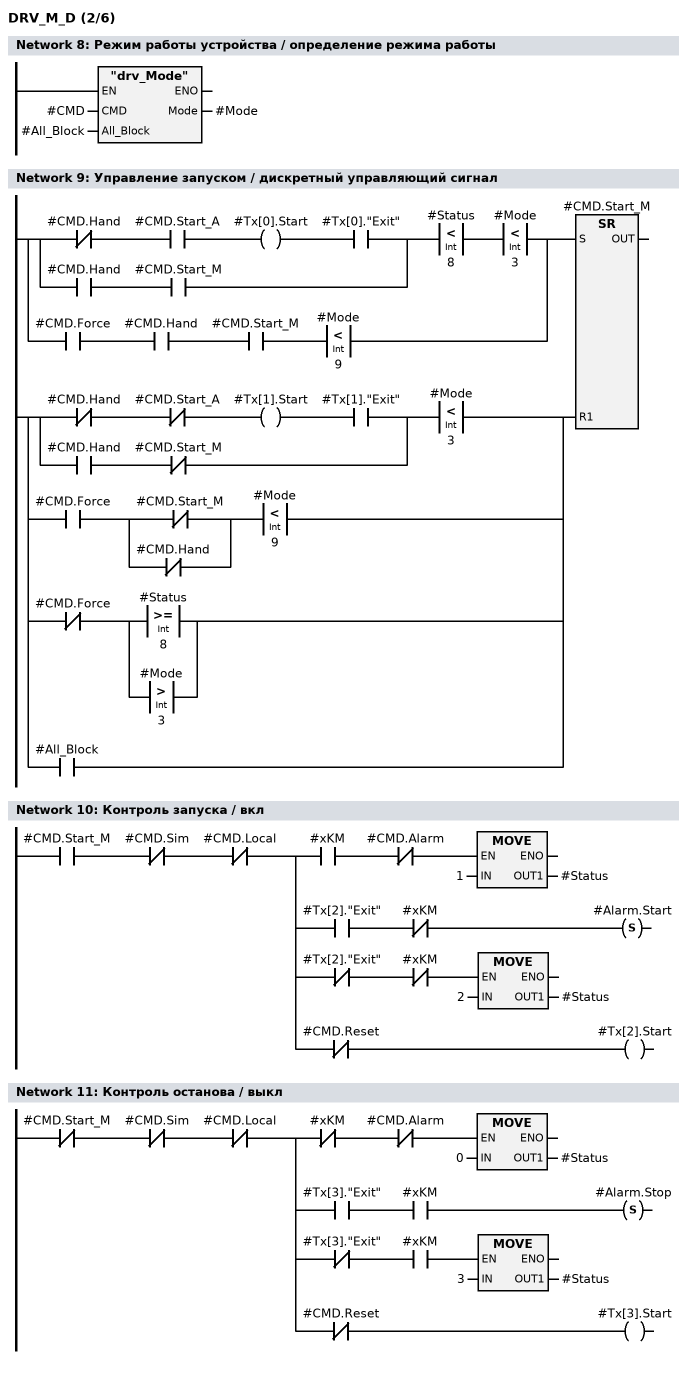
   RUNG wire#powerrail
      "drv_Mode"(CMD := #CMD, All_Block := #All_Block, Mode => #Mode)
   END_RUNG
   // the same network as SCL:
   "drv_Mode"(CMD := #CMD, All_Block := #All_Block, Mode => #Mode);
END_REGION

REGION Network 9: Управление запуском / дискретный управляющий сигнал
   RUNG wire#powerrail
      I_Contact( #CMD.Hand )
      Contact( #CMD.Start_A )
      Coil( #Tx[0].Start )
      Contact( #Tx[0]."Exit" )
      wire#w1
      { S7_Templates := "SrcType := Int" } LT_Contact(in1 := #Status, in2 := 8)
      { S7_Templates := "SrcType := Int" } LT_Contact(in1 := #Mode, in2 := 3)
      wire#w2
      S_SR(operand := #CMD.Start_M, r1 := wire#w7)
   END_RUNG
   RUNG wire#powerrail
      Contact( #CMD.Hand )
      Contact( #CMD.Start_M )
   END_RUNG wire#w1
   RUNG wire#powerrail
      Contact( #CMD.Force )
      Contact( #CMD.Hand )
      Contact( #CMD.Start_M )
      { S7_Templates := "SrcType := Int" } LT_Contact(in1 := #Mode, in2 := 9)
   END_RUNG wire#w2
   RUNG wire#powerrail
      I_Contact( #CMD.Hand )
      I_Contact( #CMD.Start_A )
      Coil( #Tx[1].Start )
      Contact( #Tx[1]."Exit" )
      wire#w3
      { S7_Templates := "SrcType := Int" } LT_Contact(in1 := #Mode, in2 := 3)
   END_RUNG wire#w7
   RUNG wire#powerrail
      Contact( #CMD.Hand )
      I_Contact( #CMD.Start_M )
   END_RUNG wire#w3
   RUNG wire#powerrail
      Contact( #CMD.Force )
      wire#w4
      I_Contact( #CMD.Start_M )
      wire#w5
      { S7_Templates := "SrcType := Int" } LT_Contact(in1 := #Mode, in2 := 9)
   END_RUNG wire#w7
   RUNG wire#w4
      I_Contact( #CMD.Hand )
   END_RUNG wire#w5
   RUNG wire#powerrail
      I_Contact( #CMD.Force )
      wire#w6
      { S7_Templates := "SrcType := Int" } GE_Contact(in1 := #Status, in2 := 8)
   END_RUNG wire#w7
   RUNG wire#w6
      { S7_Templates := "SrcType := Int" } GT_Contact(in1 := #Mode, in2 := 3)
   END_RUNG wire#w7
   RUNG wire#powerrail
      Contact( #All_Block )
   END_RUNG wire#w7
   // the same network as SCL:
   #Tx[0].Start := NOT #CMD.Hand AND #CMD.Start_A;
   #_w1 := (((NOT #CMD.Hand AND #CMD.Start_A AND #Tx[0]."Exit") OR (#CMD.Hand AND #CMD.Start_M)) AND (#Status < 8) AND (#Mode < 3)) OR (#CMD.Force AND #CMD.Hand AND #CMD.Start_M AND (#Mode < 9));
   #Tx[1].Start := NOT #CMD.Hand AND NOT #CMD.Start_A;
   #_w2 := (((NOT #CMD.Hand AND NOT #CMD.Start_A AND #Tx[1]."Exit") OR (#CMD.Hand AND NOT #CMD.Start_M)) AND (#Mode < 3)) OR (#CMD.Force AND (NOT #CMD.Start_M OR NOT #CMD.Hand) AND (#Mode < 9)) OR (NOT #CMD.Force AND ((#Status >= 8) OR (#Mode > 3))) OR #All_Block;
   IF #_w1 THEN
       #CMD.Start_M := TRUE;   // SR flip-flop
   END_IF;
   IF #_w2 THEN #CMD.Start_M := FALSE; END_IF;
END_REGION

REGION Network 10: Контроль запуска / вкл
   RUNG wire#powerrail
      Contact( #CMD.Start_M )
      I_Contact( #CMD.Sim )
      I_Contact( #CMD.Local )
      wire#w1
      Contact( #xKM )
      I_Contact( #CMD.Alarm )
      { S7_GenerateENO := "TRUE" } Move(in := 1, out1 => #Status)
   END_RUNG
   RUNG wire#w1
      Contact( #Tx[2]."Exit" )
      I_Contact( #xKM )
      S_Coil( #Alarm.Start )
   END_RUNG
   RUNG wire#w1
      I_Contact( #Tx[2]."Exit" )
      I_Contact( #xKM )
      { S7_GenerateENO := "TRUE" } Move(in := 2, out1 => #Status)
   END_RUNG
   RUNG wire#w1
      I_Contact( #CMD.Reset )
      Coil( #Tx[2].Start )
   END_RUNG
   // the same network as SCL:
   #_w1 := #CMD.Start_M AND NOT #CMD.Sim AND NOT #CMD.Local;
   IF #_w1 AND #xKM AND NOT #CMD.Alarm THEN #Status := 1; END_IF;
   IF #_w1 AND #Tx[2]."Exit" AND NOT #xKM THEN #Alarm.Start := TRUE; END_IF;
   IF #_w1 AND NOT #Tx[2]."Exit" AND NOT #xKM THEN #Status := 2; END_IF;
   #Tx[2].Start := #_w1 AND NOT #CMD.Reset;
END_REGION

REGION Network 11: Контроль останова / выкл
   RUNG wire#powerrail
      I_Contact( #CMD.Start_M )
      I_Contact( #CMD.Sim )
      I_Contact( #CMD.Local )
      wire#w1
      I_Contact( #xKM )
      I_Contact( #CMD.Alarm )
      { S7_GenerateENO := "TRUE" } Move(in := 0, out1 => #Status)
   END_RUNG
   RUNG wire#w1
      Contact( #Tx[3]."Exit" )
      Contact( #xKM )
      S_Coil( #Alarm.Stop )
   END_RUNG
   RUNG wire#w1
      I_Contact( #Tx[3]."Exit" )
      Contact( #xKM )
      { S7_GenerateENO := "TRUE" } Move(in := 3, out1 => #Status)
   END_RUNG
   RUNG wire#w1
      I_Contact( #CMD.Reset )
      Coil( #Tx[3].Start )
   END_RUNG
   // the same network as SCL:
   #_w1 := NOT #CMD.Start_M AND NOT #CMD.Sim AND NOT #CMD.Local;
   IF #_w1 AND NOT #xKM AND NOT #CMD.Alarm THEN #Status := 0; END_IF;
   IF #_w1 AND #Tx[3]."Exit" AND #xKM THEN #Alarm.Stop := TRUE; END_IF;
   IF #_w1 AND NOT #Tx[3]."Exit" AND #xKM THEN #Status := 3; END_IF;
   #Tx[3].Start := #_w1 AND NOT #CMD.Reset;
END_REGION

REGION Network 12: Локальный режим
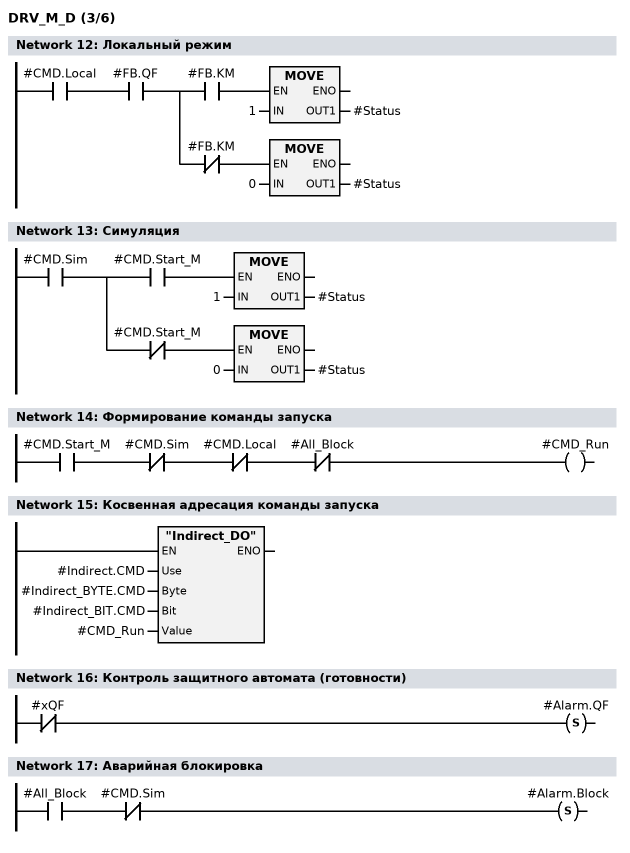
   RUNG wire#powerrail
      Contact( #CMD.Local )
      Contact( #FB.QF )
      wire#w1
      Contact( #FB.KM )
      { S7_GenerateENO := "TRUE" } Move(in := 1, out1 => #Status)
   END_RUNG
   RUNG wire#w1
      I_Contact( #FB.KM )
      { S7_GenerateENO := "TRUE" } Move(in := 0, out1 => #Status)
   END_RUNG
   // the same network as SCL:
   #_w1 := #CMD.Local AND #FB.QF;
   IF #_w1 AND #FB.KM THEN #Status := 1; END_IF;
   IF #_w1 AND NOT #FB.KM THEN #Status := 0; END_IF;
END_REGION

REGION Network 13: Симуляция
   RUNG wire#powerrail
      Contact( #CMD.Sim )
      wire#w1
      Contact( #CMD.Start_M )
      { S7_GenerateENO := "TRUE" } Move(in := 1, out1 => #Status)
   END_RUNG
   RUNG wire#w1
      I_Contact( #CMD.Start_M )
      { S7_GenerateENO := "TRUE" } Move(in := 0, out1 => #Status)
   END_RUNG
   // the same network as SCL:
   IF #CMD.Sim AND #CMD.Start_M THEN #Status := 1; END_IF;
   IF #CMD.Sim AND NOT #CMD.Start_M THEN #Status := 0; END_IF;
END_REGION

REGION Network 14: Формирование команды запуска
   RUNG wire#powerrail
      Contact( #CMD.Start_M )
      I_Contact( #CMD.Sim )
      I_Contact( #CMD.Local )
      I_Contact( #All_Block )
      Coil( #CMD_Run )
   END_RUNG
   // the same network as SCL:
   #CMD_Run := #CMD.Start_M AND NOT #CMD.Sim AND NOT #CMD.Local AND NOT #All_Block;
END_REGION

REGION Network 15: Косвенная адресация команды запуска
   RUNG wire#powerrail
      "Indirect_DO"(Use := #Indirect.CMD, "Byte" := #Indirect_BYTE.CMD, Bit := #Indirect_BIT.CMD, Value := #CMD_Run)
   END_RUNG
   // the same network as SCL:
   "Indirect_DO"(Use := #Indirect.CMD,
                 "Byte" := #Indirect_BYTE.CMD,
                 Bit := #Indirect_BIT.CMD,
                 Value := #CMD_Run);
END_REGION

REGION Network 16: Контроль защитного автомата (готовности)
   RUNG wire#powerrail
      I_Contact( #xQF )
      S_Coil( #Alarm.QF )
   END_RUNG
   // the same network as SCL:
   IF NOT #xQF THEN #Alarm.QF := TRUE; END_IF;
END_REGION

REGION Network 17: Аварийная блокировка
   RUNG wire#powerrail
      Contact( #All_Block )
      I_Contact( #CMD.Sim )
      S_Coil( #Alarm.Block )
   END_RUNG
   // the same network as SCL:
   IF #All_Block AND NOT #CMD.Sim THEN #Alarm.Block := TRUE; END_IF;
END_REGION

REGION Network 18: Сигнал аварии
   // Safety - сработал датчик безопасности, подключается через отдельный дискретный вход
   // Termo - сработала термозащита, подключается через отдельный дискретный вход
   // Alarm - сработала внешняя авария, подключается через отдельный дискретный вход
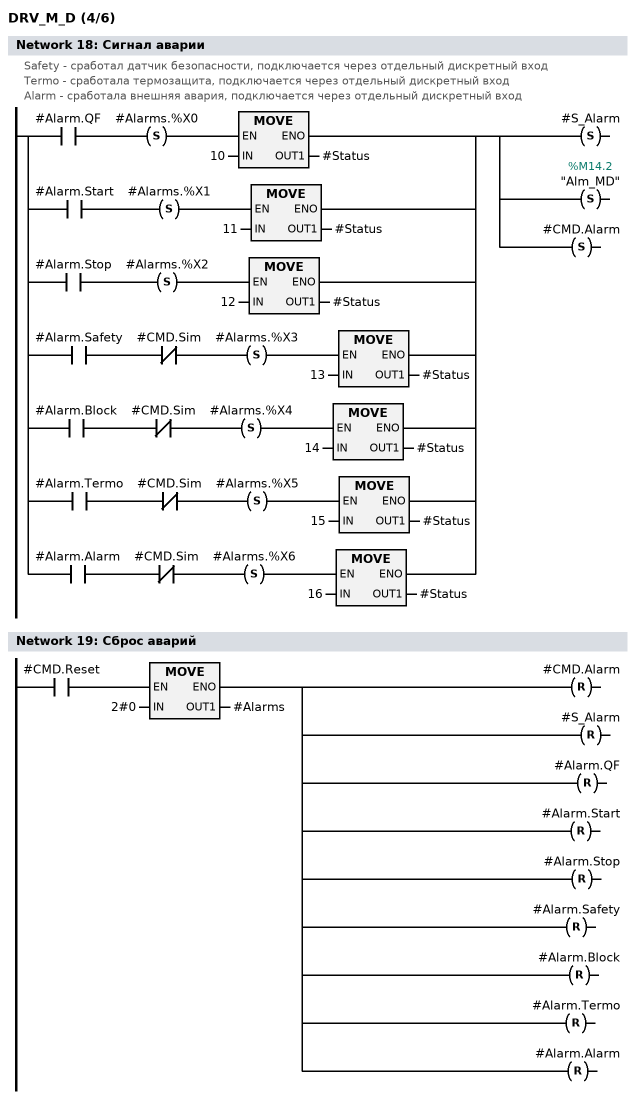
   RUNG wire#powerrail
      Contact( #Alarm.QF )
      S_Coil( #Alarms.%X0 )
      { S7_GenerateENO := "TRUE" } Move(in := 10, out1 => #Status)
      wire#w1
      S_Coil( #S_Alarm )
   END_RUNG
   RUNG wire#powerrail
      Contact( #Alarm.Start )
      S_Coil( #Alarms.%X1 )
      { S7_GenerateENO := "TRUE" } Move(in := 11, out1 => #Status)
   END_RUNG wire#w1
   RUNG wire#powerrail
      Contact( #Alarm.Stop )
      S_Coil( #Alarms.%X2 )
      { S7_GenerateENO := "TRUE" } Move(in := 12, out1 => #Status)
   END_RUNG wire#w1
   RUNG wire#powerrail
      Contact( #Alarm.Safety )
      I_Contact( #CMD.Sim )
      S_Coil( #Alarms.%X3 )
      { S7_GenerateENO := "TRUE" } Move(in := 13, out1 => #Status)
   END_RUNG wire#w1
   RUNG wire#powerrail
      Contact( #Alarm.Block )
      I_Contact( #CMD.Sim )
      S_Coil( #Alarms.%X4 )
      { S7_GenerateENO := "TRUE" } Move(in := 14, out1 => #Status)
   END_RUNG wire#w1
   RUNG wire#powerrail
      Contact( #Alarm.Termo )
      I_Contact( #CMD.Sim )
      S_Coil( #Alarms.%X5 )
      { S7_GenerateENO := "TRUE" } Move(in := 15, out1 => #Status)
   END_RUNG wire#w1
   RUNG wire#powerrail
      Contact( #Alarm.Alarm )
      I_Contact( #CMD.Sim )
      S_Coil( #Alarms.%X6 )
      { S7_GenerateENO := "TRUE" } Move(in := 16, out1 => #Status)
   END_RUNG wire#w1
   RUNG wire#w1
      S_Coil( "Alm_MD" )
   END_RUNG
   RUNG wire#w1
      S_Coil( #CMD.Alarm )
   END_RUNG
   // the same network as SCL:
   // ENO of a box is taken as its EN; it also drops when the box reports an error
   IF #Alarm.QF THEN
       #Alarms.%X0 := TRUE;
       #Status := 10;
   END_IF;
   IF #Alarm.Start THEN
       #Alarms.%X1 := TRUE;
       #Status := 11;
   END_IF;
   IF #Alarm.Stop THEN
       #Alarms.%X2 := TRUE;
       #Status := 12;
   END_IF;
   #_w1 := #Alarm.Safety AND NOT #CMD.Sim;
   IF #_w1 THEN
       #Alarms.%X3 := TRUE;
       #Status := 13;
   END_IF;
   #_w2 := #Alarm.Block AND NOT #CMD.Sim;
   IF #_w2 THEN
       #Alarms.%X4 := TRUE;
       #Status := 14;
   END_IF;
   #_w3 := #Alarm.Termo AND NOT #CMD.Sim;
   IF #_w3 THEN
       #Alarms.%X5 := TRUE;
       #Status := 15;
   END_IF;
   #_w4 := #Alarm.Alarm AND NOT #CMD.Sim;
   IF #_w4 THEN
       #Alarms.%X6 := TRUE;
       #Status := 16;
   END_IF;
   IF #Alarm.QF OR #Alarm.Start OR #Alarm.Stop OR #_w1 OR #_w2 OR #_w3 OR #_w4 THEN
       #S_Alarm := TRUE;
       "Alm_MD" := TRUE;
       #CMD.Alarm := TRUE;
   END_IF;
END_REGION

REGION Network 19: Сброс аварий
   RUNG wire#powerrail
      Contact( #CMD.Reset )
      Move(in := 2#0, out1 => #Alarms)
      wire#w1
      R_Coil( #CMD.Alarm )
   END_RUNG
   RUNG wire#w1
      R_Coil( #S_Alarm )
   END_RUNG
   RUNG wire#w1
      R_Coil( #Alarm.QF )
   END_RUNG
   RUNG wire#w1
      R_Coil( #Alarm.Start )
   END_RUNG
   RUNG wire#w1
      R_Coil( #Alarm.Stop )
   END_RUNG
   RUNG wire#w1
      R_Coil( #Alarm.Safety )
   END_RUNG
   RUNG wire#w1
      R_Coil( #Alarm.Block )
   END_RUNG
   RUNG wire#w1
      R_Coil( #Alarm.Termo )
   END_RUNG
   RUNG wire#w1
      R_Coil( #Alarm.Alarm )
   END_RUNG
   // the same network as SCL:
   IF #CMD.Reset THEN
       #Alarms := 2#0;
       #CMD.Alarm := FALSE;
       #S_Alarm := FALSE;
       #Alarm.QF := FALSE;
       #Alarm.Start := FALSE;
       #Alarm.Stop := FALSE;
       #Alarm.Safety := FALSE;
       #Alarm.Block := FALSE;
       #Alarm.Termo := FALSE;
       #Alarm.Alarm := FALSE;
   END_IF;
END_REGION

REGION Network 20: События привода
   // 0 - ручной режим активирован
   // 1 - ручной режим деактивирован
   // 2 - принудительный режим активирован
   // 3 - принудительный режим деактивирован
   // 4 - запуск в ручном режиме
   // 5 - останов в ручном режиме
   // 6 - местный режим управления активирован
   // 7 - местный режим управления деактивирован
   // 8 - запущено в местном режиме
   // 9 - остановлено в местном режиме
   // 10 - проведено сервисное обслуживание
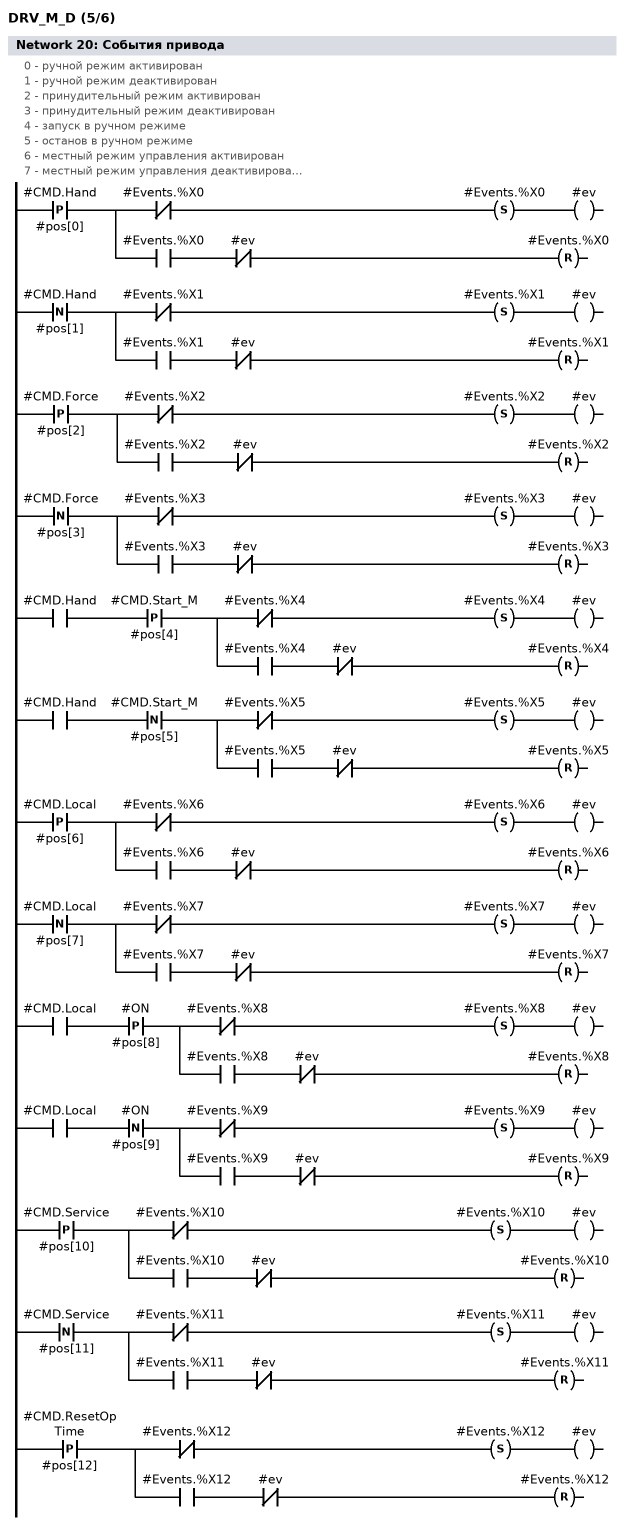
   RUNG wire#powerrail
      P_Contact(operand := #CMD.Hand, bit := #pos[0])
      wire#w1
      I_Contact( #Events.%X0 )
      S_Coil( #Events.%X0 )
      Coil( #ev )
   END_RUNG
   RUNG wire#w1
      Contact( #Events.%X0 )
      I_Contact( #ev )
      R_Coil( #Events.%X0 )
   END_RUNG
   RUNG wire#powerrail
      N_Contact(operand := #CMD.Hand, bit := #pos[1])
      wire#w2
      I_Contact( #Events.%X1 )
      S_Coil( #Events.%X1 )
      Coil( #ev )
   END_RUNG
   RUNG wire#w2
      Contact( #Events.%X1 )
      I_Contact( #ev )
      R_Coil( #Events.%X1 )
   END_RUNG
   RUNG wire#powerrail
      P_Contact(operand := #CMD.Force, bit := #pos[2])
      wire#w3
      I_Contact( #Events.%X2 )
      S_Coil( #Events.%X2 )
      Coil( #ev )
   END_RUNG
   RUNG wire#w3
      Contact( #Events.%X2 )
      I_Contact( #ev )
      R_Coil( #Events.%X2 )
   END_RUNG
   RUNG wire#powerrail
      N_Contact(operand := #CMD.Force, bit := #pos[3])
      wire#w4
      I_Contact( #Events.%X3 )
      S_Coil( #Events.%X3 )
      Coil( #ev )
   END_RUNG
   RUNG wire#w4
      Contact( #Events.%X3 )
      I_Contact( #ev )
      R_Coil( #Events.%X3 )
   END_RUNG
   RUNG wire#powerrail
      Contact( #CMD.Hand )
      P_Contact(operand := #CMD.Start_M, bit := #pos[4])
      wire#w5
      I_Contact( #Events.%X4 )
      S_Coil( #Events.%X4 )
      Coil( #ev )
   END_RUNG
   RUNG wire#w5
      Contact( #Events.%X4 )
      I_Contact( #ev )
      R_Coil( #Events.%X4 )
   END_RUNG
   RUNG wire#powerrail
      Contact( #CMD.Hand )
      N_Contact(operand := #CMD.Start_M, bit := #pos[5])
      wire#w6
      I_Contact( #Events.%X5 )
      S_Coil( #Events.%X5 )
      Coil( #ev )
   END_RUNG
   RUNG wire#w6
      Contact( #Events.%X5 )
      I_Contact( #ev )
      R_Coil( #Events.%X5 )
   END_RUNG
   RUNG wire#powerrail
      P_Contact(operand := #CMD.Local, bit := #pos[6])
      wire#w7
      I_Contact( #Events.%X6 )
      S_Coil( #Events.%X6 )
      Coil( #ev )
   END_RUNG
   RUNG wire#w7
      Contact( #Events.%X6 )
      I_Contact( #ev )
      R_Coil( #Events.%X6 )
   END_RUNG
   RUNG wire#powerrail
      N_Contact(operand := #CMD.Local, bit := #pos[7])
      wire#w8
      I_Contact( #Events.%X7 )
      S_Coil( #Events.%X7 )
      Coil( #ev )
   END_RUNG
   RUNG wire#w8
      Contact( #Events.%X7 )
      I_Contact( #ev )
      R_Coil( #Events.%X7 )
   END_RUNG
   RUNG wire#powerrail
      Contact( #CMD.Local )
      P_Contact(operand := #ON, bit := #pos[8])
      wire#w9
      I_Contact( #Events.%X8 )
      S_Coil( #Events.%X8 )
      Coil( #ev )
   END_RUNG
   RUNG wire#w9
      Contact( #Events.%X8 )
      I_Contact( #ev )
      R_Coil( #Events.%X8 )
   END_RUNG
   RUNG wire#powerrail
      Contact( #CMD.Local )
      N_Contact(operand := #ON, bit := #pos[9])
      wire#w10
      I_Contact( #Events.%X9 )
      S_Coil( #Events.%X9 )
      Coil( #ev )
   END_RUNG
   RUNG wire#w10
      Contact( #Events.%X9 )
      I_Contact( #ev )
      R_Coil( #Events.%X9 )
   END_RUNG
   RUNG wire#powerrail
      P_Contact(operand := #CMD.Service, bit := #pos[10])
      wire#w11
      I_Contact( #Events.%X10 )
      S_Coil( #Events.%X10 )
      Coil( #ev )
   END_RUNG
   RUNG wire#w11
      Contact( #Events.%X10 )
      I_Contact( #ev )
      R_Coil( #Events.%X10 )
   END_RUNG
   RUNG wire#powerrail
      N_Contact(operand := #CMD.Service, bit := #pos[11])
      wire#w12
      I_Contact( #Events.%X11 )
      S_Coil( #Events.%X11 )
      Coil( #ev )
   END_RUNG
   RUNG wire#w12
      Contact( #Events.%X11 )
      I_Contact( #ev )
      R_Coil( #Events.%X11 )
   END_RUNG
   RUNG wire#powerrail
      P_Contact(operand := #CMD.ResetOpTime, bit := #pos[12])
      wire#w13
      I_Contact( #Events.%X12 )
      S_Coil( #Events.%X12 )
      Coil( #ev )
   END_RUNG
   RUNG wire#w13
      Contact( #Events.%X12 )
      I_Contact( #ev )
      R_Coil( #Events.%X12 )
   END_RUNG
   // the same network as SCL:
   #_w1 := #CMD.Hand AND NOT #pos[0];   // rising edge of #CMD.Hand
   #pos[0] := #CMD.Hand;
   #_w2 := #_w1 AND NOT #Events.%X0;
   IF #_w2 THEN #Events.%X0 := TRUE; END_IF;
   #ev := #_w2;
   IF #_w1 AND #Events.%X0 AND NOT #ev THEN #Events.%X0 := FALSE; END_IF;
   #_w3 := NOT #CMD.Hand AND #pos[1];   // falling edge of #CMD.Hand
   #pos[1] := #CMD.Hand;
   #_w4 := #_w3 AND NOT #Events.%X1;
   IF #_w4 THEN #Events.%X1 := TRUE; END_IF;
   #ev := #_w4;
   IF #_w3 AND #Events.%X1 AND NOT #ev THEN #Events.%X1 := FALSE; END_IF;
   #_w5 := #CMD.Force AND NOT #pos[2];   // rising edge of #CMD.Force
   #pos[2] := #CMD.Force;
   #_w6 := #_w5 AND NOT #Events.%X2;
   IF #_w6 THEN #Events.%X2 := TRUE; END_IF;
   #ev := #_w6;
   IF #_w5 AND #Events.%X2 AND NOT #ev THEN #Events.%X2 := FALSE; END_IF;
   #_w7 := NOT #CMD.Force AND #pos[3];   // falling edge of #CMD.Force
   #pos[3] := #CMD.Force;
   #_w8 := #_w7 AND NOT #Events.%X3;
   IF #_w8 THEN #Events.%X3 := TRUE; END_IF;
   #ev := #_w8;
   IF #_w7 AND #Events.%X3 AND NOT #ev THEN #Events.%X3 := FALSE; END_IF;
   #_w9 := #CMD.Hand AND #CMD.Start_M AND NOT #pos[4];   // rising edge of #CMD.Start_M
   #pos[4] := #CMD.Start_M;
   #_w10 := #_w9 AND NOT #Events.%X4;
   IF #_w10 THEN #Events.%X4 := TRUE; END_IF;
   #ev := #_w10;
   IF #_w9 AND #Events.%X4 AND NOT #ev THEN #Events.%X4 := FALSE; END_IF;
   #_w11 := #CMD.Hand AND NOT #CMD.Start_M AND #pos[5];   // falling edge of #CMD.Start_M
   #pos[5] := #CMD.Start_M;
   #_w12 := #_w11 AND NOT #Events.%X5;
   IF #_w12 THEN #Events.%X5 := TRUE; END_IF;
   #ev := #_w12;
   IF #_w11 AND #Events.%X5 AND NOT #ev THEN #Events.%X5 := FALSE; END_IF;
   #_w13 := #CMD.Local AND NOT #pos[6];   // rising edge of #CMD.Local
   #pos[6] := #CMD.Local;
   #_w14 := #_w13 AND NOT #Events.%X6;
   IF #_w14 THEN #Events.%X6 := TRUE; END_IF;
   #ev := #_w14;
   IF #_w13 AND #Events.%X6 AND NOT #ev THEN #Events.%X6 := FALSE; END_IF;
   #_w15 := NOT #CMD.Local AND #pos[7];   // falling edge of #CMD.Local
   #pos[7] := #CMD.Local;
   #_w16 := #_w15 AND NOT #Events.%X7;
   IF #_w16 THEN #Events.%X7 := TRUE; END_IF;
   #ev := #_w16;
   IF #_w15 AND #Events.%X7 AND NOT #ev THEN #Events.%X7 := FALSE; END_IF;
   #_w17 := #CMD.Local AND #ON AND NOT #pos[8];   // rising edge of #ON
   #pos[8] := #ON;
   #_w18 := #_w17 AND NOT #Events.%X8;
   IF #_w18 THEN #Events.%X8 := TRUE; END_IF;
   #ev := #_w18;
   IF #_w17 AND #Events.%X8 AND NOT #ev THEN #Events.%X8 := FALSE; END_IF;
   #_w19 := #CMD.Local AND NOT #ON AND #pos[9];   // falling edge of #ON
   #pos[9] := #ON;
   #_w20 := #_w19 AND NOT #Events.%X9;
   IF #_w20 THEN #Events.%X9 := TRUE; END_IF;
   #ev := #_w20;
   IF #_w19 AND #Events.%X9 AND NOT #ev THEN #Events.%X9 := FALSE; END_IF;
   #_w21 := #CMD.Service AND NOT #pos[10];   // rising edge of #CMD.Service
   #pos[10] := #CMD.Service;
   #_w22 := #_w21 AND NOT #Events.%X10;
   IF #_w22 THEN #Events.%X10 := TRUE; END_IF;
   #ev := #_w22;
   IF #_w21 AND #Events.%X10 AND NOT #ev THEN #Events.%X10 := FALSE; END_IF;
   #_w23 := NOT #CMD.Service AND #pos[11];   // falling edge of #CMD.Service
   #pos[11] := #CMD.Service;
   #_w24 := #_w23 AND NOT #Events.%X11;
   IF #_w24 THEN #Events.%X11 := TRUE; END_IF;
   #ev := #_w24;
   IF #_w23 AND #Events.%X11 AND NOT #ev THEN #Events.%X11 := FALSE; END_IF;
   #_w25 := #CMD.ResetOpTime AND NOT #pos[12];   // rising edge of #CMD.ResetOpTime
   #pos[12] := #CMD.ResetOpTime;
   #_w26 := #_w25 AND NOT #Events.%X12;
   IF #_w26 THEN #Events.%X12 := TRUE; END_IF;
   #ev := #_w26;
   IF #_w25 AND #Events.%X12 AND NOT #ev THEN #Events.%X12 := FALSE; END_IF;
END_REGION

REGION Network 21: Сервисный режим
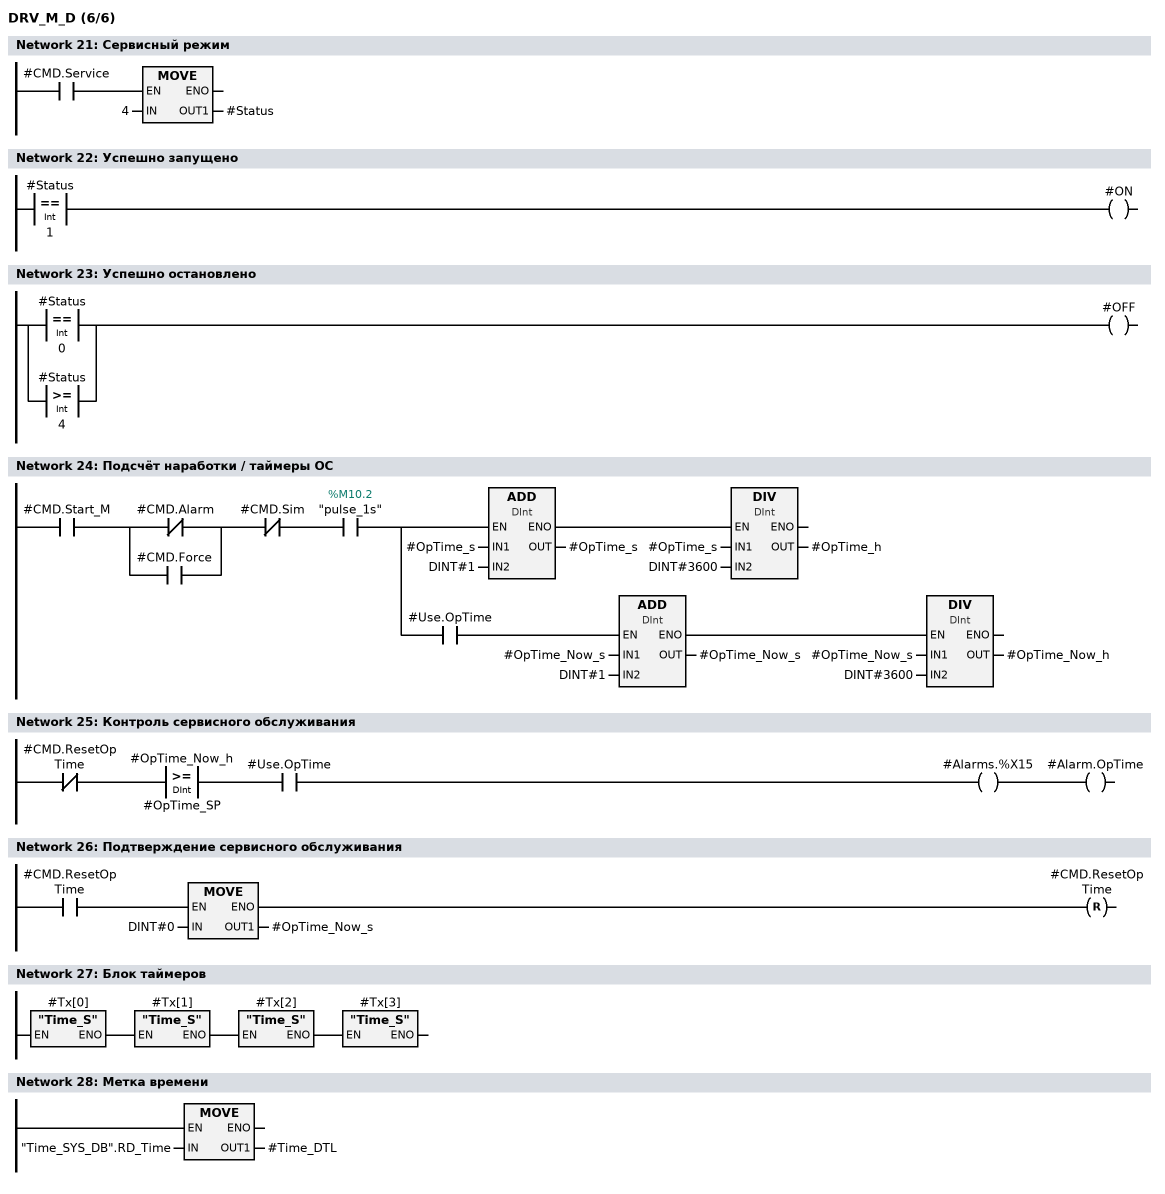
   RUNG wire#powerrail
      Contact( #CMD.Service )
      { S7_GenerateENO := "TRUE" } Move(in := 4, out1 => #Status)
   END_RUNG
   // the same network as SCL:
   IF #CMD.Service THEN #Status := 4; END_IF;
END_REGION

REGION Network 22: Успешно запущено
   RUNG wire#powerrail
      { S7_Templates := "SrcType := Int" } EQ_Contact(in1 := #Status, in2 := 1)
      Coil( #ON )
   END_RUNG
   // the same network as SCL:
   #ON := #Status = 1;
END_REGION

REGION Network 23: Успешно остановлено
   RUNG wire#powerrail
      { S7_Templates := "SrcType := Int" } EQ_Contact(in1 := #Status, in2 := 0)
      wire#w1
      Coil( #OFF )
   END_RUNG
   RUNG wire#powerrail
      { S7_Templates := "SrcType := Int" } GE_Contact(in1 := #Status, in2 := 4)
   END_RUNG wire#w1
   // the same network as SCL:
   #OFF := (#Status = 0) OR (#Status >= 4);
END_REGION

REGION Network 24: Подсчёт наработки / таймеры ОС
   RUNG wire#powerrail
      Contact( #CMD.Start_M )
      wire#w1
      I_Contact( #CMD.Alarm )
      wire#w2
      I_Contact( #CMD.Sim )
      Contact( "pulse_1s" )
      wire#w3
      { S7_Templates := "SrcType := DInt"; S7_GenerateENO := "TRUE" } Add(in1 := #OpTime_s, in2 := DINT#1, out => #OpTime_s)
      { S7_Templates := "SrcType := DInt"; S7_GenerateENO := "TRUE" } Div(in1 := #OpTime_s, in2 := DINT#3600, out => #OpTime_h)
   END_RUNG
   RUNG wire#w1
      Contact( #CMD.Force )
   END_RUNG wire#w2
   RUNG wire#w3
      Contact( #Use.OpTime )
      { S7_Templates := "SrcType := DInt"; S7_GenerateENO := "TRUE" } Add(in1 := #OpTime_Now_s, in2 := DINT#1, out => #OpTime_Now_s)
      { S7_Templates := "SrcType := DInt"; S7_GenerateENO := "TRUE" } Div(in1 := #OpTime_Now_s, in2 := DINT#3600, out => #OpTime_Now_h)
   END_RUNG
   // the same network as SCL:
   // ENO of a box is taken as its EN; it also drops when the box reports an error
   #_w1 := #CMD.Start_M AND (NOT #CMD.Alarm OR #CMD.Force) AND NOT #CMD.Sim AND "pulse_1s";
   IF #_w1 THEN
       #OpTime_s := #OpTime_s + DINT#1;
       #OpTime_h := #OpTime_s / DINT#3600;
   END_IF;
   IF #_w1 AND #Use.OpTime THEN
       #OpTime_Now_s := #OpTime_Now_s + DINT#1;
       #OpTime_Now_h := #OpTime_Now_s / DINT#3600;
   END_IF;
END_REGION

REGION Network 25: Контроль сервисного обслуживания
   RUNG wire#powerrail
      I_Contact( #CMD.ResetOpTime )
      { S7_Templates := "SrcType := DInt" } GE_Contact(in1 := #OpTime_Now_h, in2 := #OpTime_SP)
      Contact( #Use.OpTime )
      Coil( #Alarms.%X15 )
      Coil( #Alarm.OpTime )
   END_RUNG
   // the same network as SCL:
   #Alarms.%X15 := NOT #CMD.ResetOpTime AND (#OpTime_Now_h >= #OpTime_SP) AND #Use.OpTime;
   #Alarm.OpTime := #Alarms.%X15;
END_REGION

REGION Network 26: Подтверждение сервисного обслуживания
   RUNG wire#powerrail
      Contact( #CMD.ResetOpTime )
      { S7_GenerateENO := "TRUE" } Move(in := DINT#0, out1 => #OpTime_Now_s)
      R_Coil( #CMD.ResetOpTime )
   END_RUNG
   // the same network as SCL:
   // ENO of a box is taken as its EN; it also drops when the box reports an error
   IF #CMD.ResetOpTime THEN
       #OpTime_Now_s := DINT#0;
       #CMD.ResetOpTime := FALSE;
   END_IF;
END_REGION

REGION Network 27: Блок таймеров
   RUNG wire#powerrail
      #Tx[0]()
      #Tx[1]()
      #Tx[2]()
      #Tx[3]()
   END_RUNG
   // the same network as SCL:
   #Tx[0](ENO => #_w1);   // "Time_S"
   #Tx[1](EN := #_w1, ENO => #_w2);   // "Time_S"
   #Tx[2](EN := #_w2, ENO => #_w3);   // "Time_S"
   IF #_w3 THEN
       #Tx[3]();   // "Time_S"
   END_IF;
END_REGION

REGION Network 28: Метка времени
   RUNG wire#powerrail
      Move(in := "Time_SYS_DB".RD_Time, out1 => #Time_DTL)
   END_RUNG
   // the same network as SCL:
   #Time_DTL := "Time_SYS_DB".RD_Time;
END_REGION
END_FUNCTION_BLOCK

FUNCTION "drv_INV" : Void   // FC111, LAD
{ S7_Optimized_Access := 'FALSE' }
VERSION : 0.1
// stored: AutoNumber false, IsIECCheckEnabled false, SetENOAutomatically false, UDAEnableTagReadback false
   VAR_INPUT
      S : Bool;   // Сигнал
      I : Bool;   // Инверсия
   END_VAR
   VAR_IN_OUT
      R : Bool;   // Результат
   END_VAR
BEGIN

REGION Network 1: Инверсия сигнала
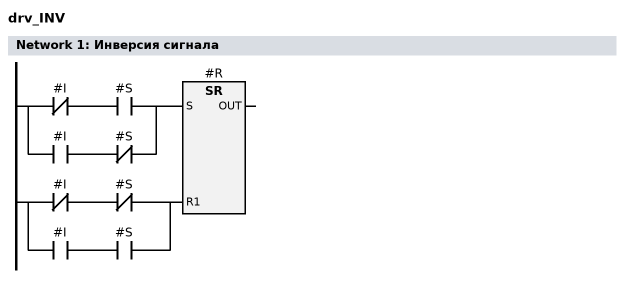
   RUNG wire#powerrail
      I_Contact( #I )
      Contact( #S )
      wire#w1
      S_SR(operand := #R, r1 := wire#w2)
   END_RUNG
   RUNG wire#powerrail
      Contact( #I )
      I_Contact( #S )
   END_RUNG wire#w1
   RUNG wire#powerrail
      I_Contact( #I )
      I_Contact( #S )
   END_RUNG wire#w2
   RUNG wire#powerrail
      Contact( #I )
      Contact( #S )
   END_RUNG wire#w2
   // the same network as SCL:
   IF (NOT #I AND #S) OR (#I AND NOT #S) THEN
       #R := TRUE;   // SR flip-flop
   END_IF;
   IF (NOT #I AND NOT #S) OR (#I AND #S) THEN #R := FALSE; END_IF;
END_REGION
END_FUNCTION

FUNCTION_BLOCK "DRV_M_DA"   // FB111, LAD
{ S7_Optimized_Access := 'FALSE' }
VERSION : 0.1
// stored: AutoNumber false, IsIECCheckEnabled false, SetENOAutomatically false, UDAEnableTagReadback false
   VAR_INPUT
      All_Block : Bool;   // Аварийный останов
   END_VAR
   VAR_IN_OUT
      FB_QF : Bool;   // защитный автомат / Защитный автомат / Готовность
      FB_KM : Bool;   // привод запущен / Пускатель / В работе
      S_Alarm : Bool;   // Внешний индикатор наличия аварии
      CMD_Run : Bool;   // Команда запуска двигателя
   END_VAR
   VAR DB_SPECIFIC
      CMD : "CMD";   // Основные команды / Блок команд
      Mode : Int;   // Режим работы
      Status : Int;   // Статус устройства
      Use : Struct   // Функционал
         QF { S7_SetPoint := 'True'} : Bool := true;   // Защитный автомат
         KM { S7_SetPoint := 'True'} : Bool := true;   // Пускатель
         OpTime { S7_SetPoint := 'True'} : Bool := true;   // Контроль наработки
         Analog { S7_SetPoint := 'True'} : Bool := true;
         Local_Keys : Bool;
      END_STRUCT;
      FB : Struct   // Функционал
         QF : Bool;   // Защитный автомат
         KM : Bool;   // Пускатель
         Local_Start : Bool;
         Local_Stop : Bool;
      END_STRUCT;
      ON : Bool;   // Успешно запущено
      OFF : Bool;   // Успешно остановлено
   END_VAR
   VAR
      Tx { S7_SetPoint := 'True'} : Array[0..3] of "Time_S";   // Блок таймеров
   END_VAR
   VAR DB_SPECIFIC
      Inv : Struct   // Инверсия сигналов
         CMD { S7_SetPoint := 'True'} : Bool;   // Команда запуска
         QF { S7_SetPoint := 'True'} : Bool;   // Защитный автомат
         KM { S7_SetPoint := 'True'} : Bool;   // Пускатель
      END_STRUCT;
      Alarm : Struct   // Сбор аварий / Список аварий
         Block : Bool;   // Аварийная остановка
         QF : Bool;   // привод не готов / Выбило защитный автомат
         Start : Bool;   // Ошибка при запуске
         Stop : Bool;   // Ошибка при останове
         Termo : Bool;   // термозащита / Сработала термозащита
         Alarm : Bool;   // Внешняя авария
         Safety : Bool;   // Сработала безопасность
         OpTime : Bool;
      END_STRUCT;
      Alarms : Word;   // Слово аварий
      Events : Word;   // События
      pos : Array[0..15] of Bool;
      OpTime_h : DInt;   // наработка (ч)
      OpTime_s { S7_SetPoint := 'True'} : DInt;   // наработка (с)
      OpTime_SP { S7_SetPoint := 'True'} : DInt := 2160;   // Интервал обслуживания, ч
      OpTime_Now_h : DInt;   // Прошло с прошлого обслуживания, ч
      OpTime_Now_s { S7_SetPoint := 'True'} : DInt;   // Прошло с прошлого обслуживания, с
      CodeID { S7_SetPoint := 'True'} : Int;   // Код датчика для привязки в скаде
      Indirect : Struct   // Использование косвенной адресации
         FB_QF { S7_SetPoint := 'True'} : Bool := true;   // защитный автомат / Защитный автомат
         FB_KM { S7_SetPoint := 'True'} : Bool := true;   // привод запущен / Пускатель
         CMD { S7_SetPoint := 'True'} : Bool := true;   // Команда запуска привода
      END_STRUCT;
      Indirect_BYTE : Struct   // Адрес входа на контроллере (Байт)
         FB_QF { S7_SetPoint := 'True'} : Int;   // защитный автомат / Защитный автомат
         FB_KM { S7_SetPoint := 'True'} : Int;   // привод запущен / Пускатель
         CMD { S7_SetPoint := 'True'} : Int;   // Команда запуска привода
      END_STRUCT;
      Indirect_BIT : Struct   // Адрес входа на контроллере (Бит)
         FB_QF { S7_SetPoint := 'True'} : Int := 9;   // защитный автомат / Защитный автомат
         FB_KM { S7_SetPoint := 'True'} : Int := 9;   // привод запущен / Пускатель
         CMD { S7_SetPoint := 'True'} : Int := 9;   // Команда запуска привода
      END_STRUCT;
      SP_A : Real;   // Уставка скорости в авторежиме
      SP_M : Real;   // Уставка скорости в ручном режиме
      ADDR { S7_SetPoint := 'True'} : Int;   // Уставка
   END_VAR
   VAR
      Converter { S7_SetPoint := 'True'} : "Converter_LAD";   // Масштабирование сигнала
   END_VAR
   VAR DB_SPECIFIC
      VmA : Real;   // Реальный сигнал на входе ПЛК
      Output_Type { S7_SetPoint := 'True'} : Int;   // Тип выхода, 0 - 4..20, 1 - 0..20, 2 - 0..10, 3 - 0..5
      "Type" { S7_SetPoint := 'True'} : Int;   // Размерность
   END_VAR
   VAR
      Slow { S7_SetPoint := 'True'} : "Slow";   // Плавный разгон и замедление
   END_VAR
   VAR DB_SPECIFIC
      Time_DTL { S7_SetPoint := 'True'} : DTL;
   END_VAR
   VAR_TEMP
      ev : Bool;
      xQF : Bool;
      xKM : Bool;
      xSP : Real;
      Signal_R : Real;   // Актуальный сигнал
      Signal_Dint : DInt;   // Сигнал в DInt
      Signal_Ex : Int;   // Конвертация сигнала
      Type_Min : Real;
      Type_Max : Real;
   END_VAR
   VAR_TEMP   // added for the SCL form of the ladder/FBD networks
      _w1 : Bool;
      _w2 : Bool;
      _w3 : Bool;
      _w4 : Bool;
      _w5 : Bool;
      _w6 : Bool;
      _w7 : Bool;
      _w8 : Bool;
      _w9 : Bool;
      _w10 : Bool;
      _w11 : Bool;
      _w12 : Bool;
      _w13 : Bool;
      _w14 : Bool;
      _w15 : Bool;
      _w16 : Bool;
      _w17 : Bool;
      _w18 : Bool;
      _w19 : Bool;
      _w20 : Bool;
      _w21 : Bool;
      _w22 : Bool;
      _w23 : Bool;
      _w24 : Bool;
      _w25 : Bool;
      _w26 : Bool;
   END_VAR
BEGIN

REGION Network 1: Режим глобальной симуляции
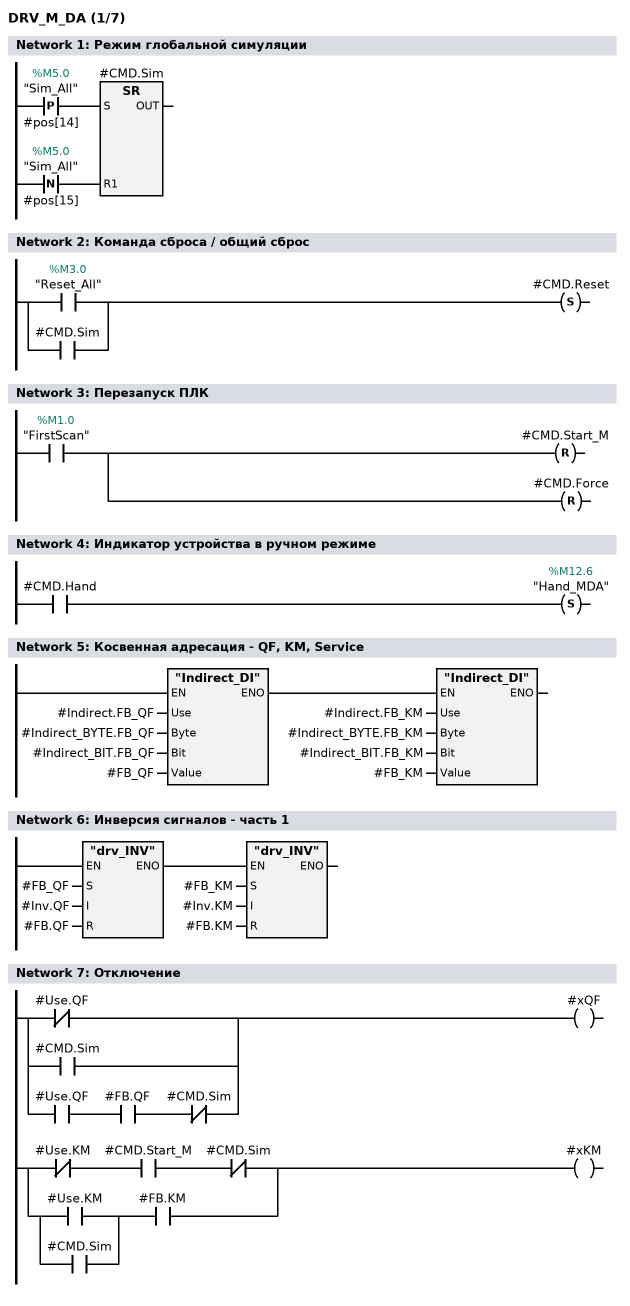
   RUNG wire#powerrail
      P_Contact(operand := "Sim_All", bit := #pos[14])
      S_SR(operand := #CMD.Sim, r1 := wire#w1)
   END_RUNG
   RUNG wire#powerrail
      N_Contact(operand := "Sim_All", bit := #pos[15])
   END_RUNG wire#w1
   // the same network as SCL:
   #_w1 := "Sim_All" AND NOT #pos[14];   // rising edge of "Sim_All"
   #pos[14] := "Sim_All";
   #_w2 := NOT "Sim_All" AND #pos[15];   // falling edge of "Sim_All"
   #pos[15] := "Sim_All";
   IF #_w1 THEN
       #CMD.Sim := TRUE;   // SR flip-flop
   END_IF;
   IF #_w2 THEN #CMD.Sim := FALSE; END_IF;
END_REGION

REGION Network 2: Команда сброса / общий сброс
   RUNG wire#powerrail
      Contact( "Reset_All" )
      wire#w1
      S_Coil( #CMD.Reset )
   END_RUNG
   RUNG wire#powerrail
      Contact( #CMD.Sim )
   END_RUNG wire#w1
   // the same network as SCL:
   IF "Reset_All" OR #CMD.Sim THEN #CMD.Reset := TRUE; END_IF;
END_REGION

REGION Network 3: Перезапуск ПЛК
   RUNG wire#powerrail
      Contact( "FirstScan" )
      wire#w1
      R_Coil( #CMD.Start_M )
   END_RUNG
   RUNG wire#w1
      R_Coil( #CMD.Force )
   END_RUNG
   // the same network as SCL:
   IF "FirstScan" THEN
       #CMD.Start_M := FALSE;
       #CMD.Force := FALSE;
   END_IF;
END_REGION

REGION Network 4: Индикатор устройства в ручном режиме
   RUNG wire#powerrail
      Contact( #CMD.Hand )
      S_Coil( "Hand_MDA" )
   END_RUNG
   // the same network as SCL:
   IF #CMD.Hand THEN "Hand_MDA" := TRUE; END_IF;
END_REGION

REGION Network 5: Косвенная адресация - QF, KM, Service
   RUNG wire#powerrail
      "Indirect_DI"(Use := #Indirect.FB_QF, "Byte" := #Indirect_BYTE.FB_QF, Bit := #Indirect_BIT.FB_QF, Value := #FB_QF)
      "Indirect_DI"(Use := #Indirect.FB_KM, "Byte" := #Indirect_BYTE.FB_KM, Bit := #Indirect_BIT.FB_KM, Value := #FB_KM)
   END_RUNG
   // the same network as SCL:
   "Indirect_DI"(Use := #Indirect.FB_QF,
                 "Byte" := #Indirect_BYTE.FB_QF,
                 Bit := #Indirect_BIT.FB_QF,
                 Value := #FB_QF,
                 ENO => #_w1);
   IF #_w1 THEN
       "Indirect_DI"(Use := #Indirect.FB_KM,
                     "Byte" := #Indirect_BYTE.FB_KM,
                     Bit := #Indirect_BIT.FB_KM,
                     Value := #FB_KM);
   END_IF;
END_REGION

REGION Network 6: Инверсия сигналов - часть 1
   RUNG wire#powerrail
      "drv_INV"(S := #FB_QF, I := #Inv.QF, R := #FB.QF)
      "drv_INV"(S := #FB_KM, I := #Inv.KM, R := #FB.KM)
   END_RUNG
   // the same network as SCL:
   "drv_INV"(S := #FB_QF, I := #Inv.QF, R := #FB.QF, ENO => #_w1);
   IF #_w1 THEN "drv_INV"(S := #FB_KM, I := #Inv.KM, R := #FB.KM); END_IF;
END_REGION

